   S_707.SPARE89 := FALSE;
   S_707.SPARE90 := FALSE;
   S_707.SPARE91 := FALSE;
   S_707.SPARE92 := FALSE;
   S_707.SPARE93 := FALSE;
   S_707.SPARE94 := FALSE;
   S_707.SPARE95 := FALSE;
   S_707.TL_DC_M_ADV_PB := FALSE;
   S_707.TL_DC_M_RET_PB := FALSE;
   S_707.SPARE98 := FALSE;
   S_707.SPARE99 := FALSE;
   S_707.SPARE100 := FALSE;
   S_707.SPARE101 := FALSE;
   S_707.SPARE102 := FALSE;
   S_707.SPARE103 := FALSE;
   S_707.SPARE104 := FALSE;
   S_707.SPARE105 := FALSE;
   S_707.SPARE106 := FALSE;
   S_707.SPARE107 := FALSE;
   S_707.SPARE108 := FALSE;
   S_707.SPARE109 := FALSE;
   S_707.SPARE110 := FALSE;
   S_707.SPARE111 := FALSE;
   S_707.SPARE112 := FALSE;
   S_707.SPARE113 := FALSE;
   S_707.SPARE114 := FALSE;
   S_707.SPARE115 := FALSE;
   S_707.SPARE116 := FALSE;
   S_707.SPARE117 := FALSE;
   S_707.SPARE118 := FALSE;
   S_707.SPARE119 := FALSE;
   S_707.SPARE120 := FALSE;
   S_707.SPARE121 := FALSE;
   S_707.SPARE122 := FALSE;
   S_707.SPARE123 := FALSE;
   S_707.SPARE124 := FALSE;
   S_707.SPARE125 := FALSE;
   S_707.SPARE126 := FALSE;
   S_707.SPARE127 := FALSE;
   S_707.SPARE128 := FALSE;
   S_707.SPARE129 := FALSE;
   S_707.SPARE130 := FALSE;
   S_707.SPARE131 := FALSE;
   S_707.SPARE132 := FALSE;
   S_707.SPARE133 := FALSE;
   S_707.SPARE134 := FALSE;
   S_707.SPARE135 := FALSE;
   S_707.SPARE136 := FALSE;
   S_707.SPARE137 := FALSE;
   S_707.SPARE138 := FALSE;
   S_707.SPARE139 := FALSE;
   S_707.SPARE140 := FALSE;
   S_707.SPARE141 := FALSE;
   S_707.SPARE142 := FALSE;
   S_707.SPARE143 := FALSE;
   S_707.SPARE144 := FALSE;
   S_707.SPARE145 := FALSE;
   S_707.SPARE146 := FALSE;
   S_707.SPARE147 := FALSE;
   S_707.SPARE148 := FALSE;
   S_707.SPARE149 := FALSE;
   S_707.SPARE150 := FALSE;
   S_707.SPARE151 := FALSE;
   S_707.SPARE152 := FALSE;
   S_707.SPARE153 := FALSE;
   S_707.SPARE154 := FALSE;
   S_707.SPARE155 := FALSE;
   S_707.SPARE156 := FALSE;
   S_707.SPARE157 := FALSE;
   S_707.SPARE158 := FALSE;
   S_707.SPARE159 := FALSE;
   S_707.SPARE160 := FALSE;
   S_707.SPARE161 := FALSE;
   S_707.HOOK_PIN_UP_LP := W#16#0;
   S_707.HOOK_PIN_DOWN_LP := W#16#700;
   S_707.DAECHA_LOCK_ADV_LP := W#16#300;
   S_707.DAECHA_LOCK_RET_LP := W#16#0;
   S_707.ELE_ADV_LP := W#16#300;
   S_707.ELE_RET_LP := W#16#0;
   S_707.AIR_ELE_ADV_LP := W#16#300;
   S_707.AIR_ELE_RET_LP := W#16#0;
   S_707.SP_WORD19 := W#16#0;
   S_707.SP_WORD20 := W#16#0;
   S_707.LM_DC_PIN_UP_LP := W#16#0;
   S_707.LM_DC_PIN_DOWN_LP := W#16#0;
   S_707.LM_DC_1ST_CLAMP1_ADV_LP := W#16#0;
   S_707.LM_DC_1ST_CLAMP1_RET_LP := W#16#0;
   S_707.LM_DC_1ST_CLAMP2_ADV_LP := W#16#0;
   S_707.LM_DC_1ST_CLAMP2_RET_LP := W#16#0;
   S_707.LM_DC_1ST_CLAMP3_ADV_LP := W#16#0;
   S_707.LM_DC_1ST_CLAMP3_RET_LP := W#16#0;
   S_707.LM_DC_1ST_CLAMP4_ADV_LP := W#16#0;
   S_707.LM_DC_1ST_CLAMP4_RET_LP := W#16#0;
   S_707.LM_DC_2ND_CLAMP1_ADV_LP := W#16#0;
   S_707.LM_DC_2ND_CLAMP1_RET_LP := W#16#0;
   S_707.LM_DC_2ND_CLAMP2_ADV_LP := W#16#0;
   S_707.LM_DC_2ND_CLAMP2_RET_LP := W#16#0;
   S_707.LM_DC_2ND_CLAMP3_ADV_LP := W#16#0;
   S_707.LM_DC_2ND_CLAMP3_RET_LP := W#16#0;
   S_707.LM_DC_2ND_CLAMP4_ADV_LP := W#16#0;
   S_707.LM_DC_2ND_CLAMP4_RET_LP := W#16#0;
   S_707.LM_DC_2ND_CLAMP5_ADV_LP := W#16#0;
   S_707.LM_DC_2ND_CLAMP5_RET_LP := W#16#0;
   S_707.LM_DC_DR_STK_PIN_UP_LP := W#16#0;
   S_707.LM_DC_DR_STK_PIN_DOWN_LP := W#16#0;
   S_707.LM_DC_OTR_CLAMP_ADV_LP := W#16#0;
   S_707.LM_DC_OTR_CLAMP_RET_LP := W#16#0;
   S_707.LM_DC_ASSY_CLAMP_ADV_LP := W#16#0;
   S_707.LM_DC_ASSY_CLAMP_RET_LP := W#16#0;
   S_707.LM_DC_FF_PIN_UP_LP := W#16#0;
   S_707.LM_DC_FF_PIN_DOWN_LP := W#16#0;
   S_707.LM_DC_FF_CLAMP_ADV_LP := W#16#0;
   S_707.LM_DC_FF_CLAMP_RET_LP := W#16#0;
   S_707.LM_DC_2ND_CLAMP6_ADV_LP := W#16#0;
   S_707.LM_DC_2ND_CLAMP6_RET_LP := W#16#0;
   S_707.LM_DC_2ND_CLAMP7_ADV_LP := W#16#0;
   S_707.LM_DC_2ND_CLAMP7_RET_LP := W#16#0;
   S_707.LM_DC_1ST_CLAMP5_ADV_LP := W#16#0;
   S_707.LM_DC_1ST_CLAMP5_RET_LP := W#16#0;
   S_707.SP_WORD68 := W#16#0;
   S_707.SP_WORD69 := W#16#0;
   S_707.SP_WORD70 := W#16#0;
   S_707.SP_WORD71 := W#16#0;
   S_707.TL_DC_PIN_UP_LP := W#16#F00;
   S_707.TL_DC_PIN_DOWN_LP := W#16#0;
   S_707.TL_DC_LATCH1_ADV_LP := W#16#3F00;
   S_707.TL_DC_LATCH1_RET_LP := W#16#0;
   S_707.TL_DC_LATCH2_ADV_LP := W#16#700;
   S_707.TL_DC_LATCH2_RET_LP := W#16#0;
   S_707.TL_DC_1ST_CLAMP1_ADV_LP := W#16#300;
   S_707.TL_DC_1ST_CLAMP1_RET_LP := W#16#0;
   S_707.TL_DC_1ST_CLAMP2_ADV_LP := W#16#300;
   S_707.TL_DC_1ST_CLAMP2_RET_LP := W#16#0;
   S_707.TL_DC_1ST_CLAMP3_ADV_LP := W#16#300;
   S_707.TL_DC_1ST_CLAMP3_RET_LP := W#16#0;
   S_707.TL_DC_2ND_CLAMP1_ADV_LP := W#16#300;
   S_707.TL_DC_2ND_CLAMP1_RET_LP := W#16#0;
   S_707.TL_DC_2ND_CLAMP2_ADV_LP := W#16#300;
   S_707.TL_DC_2ND_CLAMP2_RET_LP := W#16#0;
   S_707.TL_DC_U261_ADV_LP := W#16#300;
   S_707.TL_DC_U261_RET_LP := W#16#0;
   S_707.TL_DC_U261_CLAMP_ADV_LP := W#16#300;
   S_707.TL_DC_U261_CLAMP_RET_LP := W#16#0;
   S_707.TL_DC_U269_UP_LP := W#16#100;
   S_707.TL_DC_U269_DOWN_LP := W#16#0;
   S_707.TL_DC_U269_CLAMP_ADV_LP := W#16#300;
   S_707.TL_DC_U269_CLAMP_RET_LP := W#16#0;
   S_707.TL_DC_3RD_CLAMP_ADV_LP := W#16#100;
   S_707.TL_DC_3RD_CLAMP_RET_LP := W#16#0;
   S_707.TL_DC_U262_1_UP_LP := W#16#0;
   S_707.TL_DC_U262_1_DOWN_LP := W#16#300;
   S_707.TL_DC_U262_1_ADV_LP := W#16#0;
   S_707.TL_DC_U262_1_RET_LP := W#16#300;
   S_707.TL_DC_U262_1_CLP_ADV_LP := W#16#0;
   S_707.TL_DC_U262_1_CLP_RET_LP := W#16#300;
   S_707.TL_DC_U261_2_CLP_ADV_LP := W#16#0;
   S_707.TL_DC_U261_2_CLP_RET_LP := W#16#300;
   S_707.SP_WORD106 := W#16#0;
   S_707.SP_WORD107 := W#16#0;
   S_707.SP_WORD108 := W#16#0;
   S_707.SP_WORD109 := W#16#0;
   S_707.SP_WORD110 := W#16#0;
   S_707.SP_WORD111 := W#16#0;
   S_708.M_AUTO_SEL := FALSE;
   S_708.M_MANUAL_SEL := FALSE;
   S_708.M_READY_PB := FALSE;
   S_708.M_AUTO_RUN_PB := FALSE;
   S_708.M_WORK_COMP_SET_PB := FALSE;
   S_708.M_WORK_COMP_RST_PB := FALSE;
   S_708.M_HOME_POS_PB := FALSE;
   S_708.M_708_L_R_BT_ERR_RST := FALSE;
   S_708.HOOK_PIN_SEL := FALSE;
   S_708.EJECT_SEL := FALSE;
   S_708.SAFETY_PIN_SEL := FALSE;
   S_708.DAECHA_OUT_SEL := FALSE;
   S_708.ELE_UP_DN_SEL := FALSE;
   S_708.ELE_ADV_RET_SEL := FALSE;
   S_708.SPARE15 := FALSE;
   S_708.SPARE16 := FALSE;
   S_708.SPARE17 := FALSE;
   S_708.SPARE18 := FALSE;
   S_708.SPARE19 := FALSE;
   S_708.SPARE20 := FALSE;
   S_708.SPARE21 := FALSE;
   S_708.SPARE22 := FALSE;
   S_708.SPARE23 := FALSE;
   S_708.SPARE24 := FALSE;
   S_708.SPARE25 := FALSE;
   S_708.SPARE26 := FALSE;
   S_708.SPARE27 := FALSE;
   S_708.SPARE28 := FALSE;
   S_708.SPARE29 := FALSE;
   S_708.SPARE30 := FALSE;
   S_708.M_ADV_PB := FALSE;
   S_708.M_RET_PB := FALSE;
   S_708.LM_DC_PIN_SEL := FALSE;
   S_708.LM_DC_1ST_CLAMP1_SEL := FALSE;
   S_708.LM_DC_1ST_CLAMP2_SEL := FALSE;
   S_708.LM_DC_1ST_CLAMP3_SEL := FALSE;
   S_708.LM_DC_1ST_CLAMP4_SEL := FALSE;
   S_708.LM_DC_2ND_CLAMP1_SEL := FALSE;
   S_708.LM_DC_2ND_CLAMP2_SEL := FALSE;
   S_708.LM_DC_2ND_CLAMP3_SEL := FALSE;
   S_708.LM_DC_2ND_CLAMP4_SEL := FALSE;
   S_708.LM_DC_2ND_CLAMP5_SEL := FALSE;
   S_708.LM_DC_DR_STK_PIN_SEL := FALSE;
   S_708.LM_DC_OTR_CLAMP_SEL := FALSE;
   S_708.LM_DC_ASSY_CLAMP_SEL := FALSE;
   S_708.LM_DC_FF_PIN_SEL := FALSE;
   S_708.LM_DC_FF_CLAMP_SEL := FALSE;
   S_708.LM_DC_2ND_CLAMP6_SEL := FALSE;
   S_708.SPARE50 := FALSE;
   S_708.SPARE51 := FALSE;
   S_708.SPARE52 := FALSE;
   S_708.SPARE53 := FALSE;
   S_708.SPARE54 := FALSE;
   S_708.SPARE55 := FALSE;
   S_708.SPARE56 := FALSE;
   S_708.SPARE57 := FALSE;
   S_708.SPARE58 := FALSE;
   S_708.SPARE59 := FALSE;
   S_708.SPARE60 := FALSE;
   S_708.SPARE61 := FALSE;
   S_708.SPARE62 := FALSE;
   S_708.SPARE63 := FALSE;
   S_708.LM_DC_M_ADV_PB := FALSE;
   S_708.LM_DC_M_RET_PB := FALSE;
   S_708.TL_DC_PIN_SEL := FALSE;
   S_708.TL_DC_LATCH1_SEL := FALSE;
   S_708.TL_DC_1ST_CLAMP_SEL := FALSE;
   S_708.TL_DC_2ND_CLAMP_SEL := FALSE;
   S_708.TL_DC_U261_SEL := FALSE;
   S_708.TL_DC_U261_CLAMP_SEL := FALSE;
   S_708.TL_DC_U269_UP_DN_SEL := FALSE;
   S_708.TL_DC_U269_CLAMP_SEL := FALSE;
   S_708.TL_DC_3RD_CLAMP_SEL := FALSE;
   S_708.TL_DC_U262_1_UP_DN_SEL := FALSE;
   S_708.TL_DC_U262_1_SEL := FALSE;
   S_708.TL_DC_U262_1_CLAMP_SEL := FALSE;
   S_708.TL_DC_U261_2_CLAMP_SEL := FALSE;
   S_708.SPARE79 := FALSE;
   S_708.SPARE80 := FALSE;
   S_708.SPARE81 := FALSE;
   S_708.SPARE82 := FALSE;
   S_708.SPARE83 := FALSE;
   S_708.SPARE84 := FALSE;
   S_708.SPARE85 := FALSE;
   S_708.SPARE86 := FALSE;
   S_708.SPARE87 := FALSE;
   S_708.SPARE88 := FALSE;
   S_708.SPARE89 := FALSE;
   S_708.SPARE90 := FALSE;
   S_708.SPARE91 := FALSE;
   S_708.SPARE92 := FALSE;
   S_708.SPARE93 := FALSE;
   S_708.SPARE94 := FALSE;
   S_708.SPARE95 := FALSE;
   S_708.TL_DC_M_ADV_PB := FALSE;
   S_708.TL_DC_M_RET_PB := FALSE;
   S_708.SPARE98 := FALSE;
   S_708.SPARE99 := FALSE;
   S_708.SPARE100 := FALSE;
   S_708.SPARE101 := FALSE;
   S_708.SPARE102 := FALSE;
   S_708.SPARE103 := FALSE;
   S_708.SPARE104 := FALSE;
   S_708.SPARE105 := FALSE;
   S_708.SPARE106 := FALSE;
   S_708.SPARE107 := FALSE;
   S_708.SPARE108 := FALSE;
   S_708.SPARE109 := FALSE;
   S_708.SPARE110 := FALSE;
   S_708.SPARE111 := FALSE;
   S_708.SPARE112 := FALSE;
   S_708.SPARE113 := FALSE;
   S_708.SPARE114 := FALSE;
   S_708.SPARE115 := FALSE;
   S_708.SPARE116 := FALSE;
   S_708.SPARE117 := FALSE;
   S_708.SPARE118 := FALSE;
   S_708.SPARE119 := FALSE;
   S_708.SPARE120 := FALSE;
   S_708.SPARE121 := FALSE;
   S_708.SPARE122 := FALSE;
   S_708.SPARE123 := FALSE;
   S_708.SPARE124 := FALSE;
   S_708.SPARE125 := FALSE;
   S_708.SPARE126 := FALSE;
   S_708.SPARE127 := FALSE;
   S_708.SPARE128 := FALSE;
   S_708.SPARE129 := FALSE;
   S_708.ELE_AR_ADV_LP := W#16#300;
   S_708.ELE_AR_RET_LP := W#16#0;
   S_708.HOOK_PIN_UP_LP := W#16#0;
   S_708.HOOK_PIN_DOWN_LP := W#16#300;
   S_708.EJECT_UP_LP := W#16#0;
   S_708.EJECT_DOWN_LP := W#16#300;
   S_708.SAFETY_PIN_UP_LP := W#16#300;
   S_708.SAFETY_PIN_UDOWN_LP := W#16#0;
   S_708.DAECHA_OUT_ADV_LP := W#16#0;
   S_708.DAECHA_OUT_RET_LP := W#16#0;
   S_708.ELE_UD_UP_LP := W#16#300;
   S_708.ELE_UD_DOWN_LP := W#16#0;
   S_708.LM_DC_PIN_UP_LP := W#16#0;
   S_708.LM_DC_PIN_DOWN_LP := W#16#0;
   S_708.LM_DC_1ST_CLAMP1_ADV_LP := W#16#0;
   S_708.LM_DC_1ST_CLAMP1_RET_LP := W#16#0;
   S_708.LM_DC_1ST_CLAMP2_ADV_LP := W#16#0;
   S_708.LM_DC_1ST_CLAMP2_RET_LP := W#16#0;
   S_708.LM_DC_1ST_CLAMP3_ADV_LP := W#16#0;
   S_708.LM_DC_1ST_CLAMP3_RET_LP := W#16#0;
   S_708.LM_DC_1ST_CLAMP4_ADV_LP := W#16#0;
   S_708.LM_DC_1ST_CLAMP4_RET_LP := W#16#0;
   S_708.LM_DC_2ND_CLAMP1_ADV_LP := W#16#0;
   S_708.LM_DC_2ND_CLAMP1_RET_LP := W#16#0;
   S_708.LM_DC_2ND_CLAMP2_ADV_LP := W#16#0;
   S_708.LM_DC_2ND_CLAMP2_RET_LP := W#16#0;
   S_708.LM_DC_2ND_CLAMP3_ADV_LP := W#16#0;
   S_708.LM_DC_2ND_CLAMP3_RET_LP := W#16#0;
   S_708.LM_DC_2ND_CLAMP4_ADV_LP := W#16#0;
   S_708.LM_DC_2ND_CLAMP4_RET_LP := W#16#0;
   S_708.LM_DC_2ND_CLAMP5_ADV_LP := W#16#0;
   S_708.LM_DC_2ND_CLAMP5_RET_LP := W#16#0;
   S_708.LM_DC_DR_STK_PIN_UP_LP := W#16#0;
   S_708.LM_DC_DR_STK_PIN_DOWN_LP := W#16#0;
   S_708.LM_DC_OTR_CLAMP_ADV_LP := W#16#0;
   S_708.LM_DC_OTR_CLAMP_RET_LP := W#16#0;
   S_708.LM_DC_ASSY_CLAMP_ADV_LP := W#16#0;
   S_708.LM_DC_ASSY_CLAMP_RET_LP := W#16#0;
   S_708.LM_DC_FF_PIN_UP_LP := W#16#0;
   S_708.LM_DC_FF_PIN_DOWN_LP := W#16#0;
   S_708.LM_DC_FF_CLAMP_ADV_LP := W#16#0;
   S_708.LM_DC_FF_CLAMP_RET_LP := W#16#0;
   S_708.LM_DC_2ND_CLAMP6_ADV_LP := W#16#0;
   S_708.LM_DC_2ND_CLAMP6_RET_LP := W#16#0;
   S_708.LM_DC_2ND_CLAMP7_ADV_LP := W#16#0;
   S_708.LM_DC_2ND_CLAMP7_RET_LP := W#16#0;
   S_708.LM_DC_1ST_CLAMP5_ADV_LP := W#16#0;
   S_708.LM_DC_1ST_CLAMP5_RET_LP := W#16#0;
   S_708.SP_WORD68 := W#16#0;
   S_708.SP_WORD69 := W#16#0;
   S_708.SP_WORD70 := W#16#0;
   S_708.SP_WORD71 := W#16#0;
   S_708.TL_DC_PIN_UP_LP := W#16#0;
   S_708.TL_DC_PIN_DOWN_LP := W#16#F00;
   S_708.TL_DC_LATCH1_ADV_LP := W#16#0;
   S_708.TL_DC_LATCH1_RET_LP := W#16#3F00;
   S_708.TL_DC_LATCH2_ADV_LP := W#16#0;
   S_708.TL_DC_LATCH2_RET_LP := W#16#700;
   S_708.TL_DC_1ST_CLAMP1_ADV_LP := W#16#0;
   S_708.TL_DC_1ST_CLAMP1_RET_LP := W#16#3F00;
   S_708.TL_DC_1ST_CLAMP2_ADV_LP := W#16#0;
   S_708.TL_DC_1ST_CLAMP2_RET_LP := W#16#3F00;
   S_708.TL_DC_1ST_CLAMP3_ADV_LP := W#16#0;
   S_708.TL_DC_1ST_CLAMP3_RET_LP := W#16#F00;
   S_708.TL_DC_2ND_CLAMP1_ADV_LP := W#16#0;
   S_708.TL_DC_2ND_CLAMP1_RET_LP := W#16#3F00;
   S_708.TL_DC_2ND_CLAMP2_ADV_LP := W#16#0;
   S_708.TL_DC_2ND_CLAMP2_RET_LP := W#16#3F00;
   S_708.TL_DC_U261_ADV_LP := W#16#0;
   S_708.TL_DC_U261_RET_LP := W#16#300;
   S_708.TL_DC_U261_CLAMP_ADV_LP := W#16#0;
   S_708.TL_DC_U261_CLAMP_RET_LP := W#16#300;
   S_708.TL_DC_U269_UP_LP := W#16#0;
   S_708.TL_DC_U269_DOWN_LP := W#16#300;
   S_708.TL_DC_U269_CLAMP_ADV_LP := W#16#0;
   S_708.TL_DC_U269_CLAMP_RET_LP := W#16#700;
   S_708.TL_DC_3RD_CLAMP_ADV_LP := W#16#0;
   S_708.TL_DC_3RD_CLAMP_RET_LP := W#16#300;
   S_708.TL_DC_U262_1_UP_LP := W#16#0;
   S_708.TL_DC_U262_1_DOWN_LP := W#16#300;
   S_708.TL_DC_U262_1_ADV_LP := W#16#0;
   S_708.TL_DC_U262_1_RET_LP := W#16#300;
   S_708.TL_DC_U262_1_CLP_ADV_LP := W#16#0;
   S_708.TL_DC_U262_1_CLP_RET_LP := W#16#300;
   S_708.TL_DC_U261_2_CLP_ADV_LP := W#16#0;
   S_708.TL_DC_U261_2_CLP_RET_LP := W#16#300;
   S_708.SP_WORD106 := W#16#0;
   S_708.SP_WORD107 := W#16#0;
   S_708.SP_WORD108 := W#16#0;
   S_708.SP_WORD109 := W#16#0;
   S_708.AIR_ELE_AR_ADV_LP := W#16#300;
   S_708.AIR_ELE_AR_RET_LP := W#16#0;
   S_UPDL.M_AUTO_SEL := FALSE;
   S_UPDL.M_MANUAL_SEL := FALSE;
   S_UPDL.M_READY_PB := FALSE;
   S_UPDL.M_AUTO_RUN_PB := FALSE;
   S_UPDL.M_WORK_COMP_SET_PB := FALSE;
   S_UPDL.M_WORK_COMP_RST_PB := FALSE;
   S_UPDL.M_HOME_POS_PB := FALSE;
   S_UPDL.SPARE8 := FALSE;
   S_UPDL.DAECHA_CLAMP_SEL := FALSE;
   S_UPDL.ELE_AIR_UP_DN_SEL := FALSE;
   S_UPDL.ELE_AIR_ADV_RET_SEL := FALSE;
   S_UPDL.DAECHA_IN_SEL := TRUE;
   S_UPDL.DAECHA_OUT_SEL := FALSE;
   S_UPDL.LIFT_LOCK_SEL := FALSE;
   S_UPDL.LIFT_UP_DN_SEL := FALSE;
   S_UPDL.SPARE16 := FALSE;
   S_UPDL.SPARE17 := FALSE;
   S_UPDL.SPARE18 := FALSE;
   S_UPDL.SPARE19 := FALSE;
   S_UPDL.SPARE20 := FALSE;
   S_UPDL.SPARE21 := FALSE;
   S_UPDL.SPARE22 := FALSE;
   S_UPDL.SPARE23 := FALSE;
   S_UPDL.SPARE24 := FALSE;
   S_UPDL.SPARE25 := FALSE;
   S_UPDL.SPARE26 := FALSE;
   S_UPDL.SPARE27 := FALSE;
   S_UPDL.SPARE28 := FALSE;
   S_UPDL.SPARE29 := FALSE;
   S_UPDL.SPARE30 := FALSE;
   S_UPDL.M_ADV_PB := FALSE;
   S_UPDL.M_RET_PB := FALSE;
   S_UPDL.SPARE34 := FALSE;
   S_UPDL.SPARE35 := FALSE;
   S_UPDL.SPARE36 := FALSE;
   S_UPDL.SPARE37 := FALSE;
   S_UPDL.SPARE38 := FALSE;
   S_UPDL.SPARE39 := FALSE;
   S_UPDL.SPARE40 := FALSE;
   S_UPDL.SPARE41 := FALSE;
   S_UPDL.SPARE42 := FALSE;
   S_UPDL.SPARE43 := FALSE;
   S_UPDL.SPARE44 := FALSE;
   S_UPDL.SPARE45 := FALSE;
   S_UPDL.SPARE46 := FALSE;
   S_UPDL.SPARE47 := FALSE;
   S_UPDL.SPARE48 := FALSE;
   S_UPDL.SPARE49 := FALSE;
   S_UPDL.SPARE50 := FALSE;
   S_UPDL.SPARE51 := FALSE;
   S_UPDL.SPARE52 := FALSE;
   S_UPDL.SPARE53 := FALSE;
   S_UPDL.SPARE54 := FALSE;
   S_UPDL.SPARE55 := FALSE;
   S_UPDL.SPARE56 := FALSE;
   S_UPDL.SPARE57 := FALSE;
   S_UPDL.SPARE58 := FALSE;
   S_UPDL.SPARE59 := FALSE;
   S_UPDL.SPARE60 := FALSE;
   S_UPDL.SPARE61 := FALSE;
   S_UPDL.SPARE62 := FALSE;
   S_UPDL.SPARE63 := FALSE;
   S_UPDL.SPARE64 := FALSE;
   S_UPDL.SPARE65 := FALSE;
   S_UPDL.SPARE66 := FALSE;
   S_UPDL.SPARE67 := FALSE;
   S_UPDL.SPARE68 := FALSE;
   S_UPDL.SPARE69 := FALSE;
   S_UPDL.SPARE70 := FALSE;
   S_UPDL.SPARE71 := FALSE;
   S_UPDL.SPARE72 := FALSE;
   S_UPDL.SPARE73 := FALSE;
   S_UPDL.SPARE74 := FALSE;
   S_UPDL.SPARE75 := FALSE;
   S_UPDL.SPARE76 := FALSE;
   S_UPDL.SPARE77 := FALSE;
   S_UPDL.SPARE78 := FALSE;
   S_UPDL.SPARE79 := FALSE;
   S_UPDL.SPARE80 := FALSE;
   S_UPDL.SPARE81 := FALSE;
   S_UPDL.SPARE82 := FALSE;
   S_UPDL.SPARE83 := FALSE;
   S_UPDL.SPARE84 := FALSE;
   S_UPDL.SPARE85 := FALSE;
   S_UPDL.SPARE86 := FALSE;
   S_UPDL.SPARE87 := FALSE;
   S_UPDL.SPARE88 := FALSE;
   S_UPDL.SPARE89 := FALSE;
   S_UPDL.SPARE90 := FALSE;
   S_UPDL.SPARE91 := FALSE;
   S_UPDL.SPARE92 := FALSE;
   S_UPDL.SPARE93 := FALSE;
   S_UPDL.SPARE94 := FALSE;
   S_UPDL.SPARE95 := FALSE;
   S_UPDL.SPARE96 := FALSE;
   S_UPDL.SPARE97 := FALSE;
   S_UPDL.SPARE98 := FALSE;
   S_UPDL.SPARE99 := FALSE;
   S_UPDL.SPARE100 := FALSE;
   S_UPDL.SPARE101 := FALSE;
   S_UPDL.SPARE102 := FALSE;
   S_UPDL.SPARE103 := FALSE;
   S_UPDL.SPARE104 := FALSE;
   S_UPDL.SPARE105 := FALSE;
   S_UPDL.SPARE106 := FALSE;
   S_UPDL.SPARE107 := FALSE;
   S_UPDL.SPARE108 := FALSE;
   S_UPDL.SPARE109 := FALSE;
   S_UPDL.SPARE110 := FALSE;
   S_UPDL.SPARE111 := FALSE;
   S_UPDL.SPARE112 := FALSE;
   S_UPDL.SPARE113 := FALSE;
   S_UPDL.SPARE114 := FALSE;
   S_UPDL.SPARE115 := FALSE;
   S_UPDL.SPARE116 := FALSE;
   S_UPDL.SPARE117 := FALSE;
   S_UPDL.SPARE118 := FALSE;
   S_UPDL.SPARE119 := FALSE;
   S_UPDL.SPARE120 := FALSE;
   S_UPDL.SPARE121 := FALSE;
   S_UPDL.SPARE122 := FALSE;
   S_UPDL.SPARE123 := FALSE;
   S_UPDL.SPARE124 := FALSE;
   S_UPDL.SPARE125 := FALSE;
   S_UPDL.SPARE126 := FALSE;
   S_UPDL.SPARE127 := FALSE;
   S_UPDL.SPARE128 := FALSE;
   S_UPDL.SPARE129 := FALSE;
   S_UPDL.SPARE130 := FALSE;
   S_UPDL.SPARE131 := FALSE;
   S_UPDL.SPARE132 := FALSE;
   S_UPDL.SPARE133 := FALSE;
   S_UPDL.SPARE134 := FALSE;
   S_UPDL.SPARE135 := FALSE;
   S_UPDL.SPARE136 := FALSE;
   S_UPDL.SPARE137 := FALSE;
   S_UPDL.SPARE138 := FALSE;
   S_UPDL.SPARE139 := FALSE;
   S_UPDL.SPARE140 := FALSE;
   S_UPDL.SPARE141 := FALSE;
   S_UPDL.SPARE142 := FALSE;
   S_UPDL.SPARE143 := FALSE;
   S_UPDL.SPARE144 := FALSE;
   S_UPDL.SPARE145 := FALSE;
   S_UPDL.SPARE146 := FALSE;
   S_UPDL.SPARE147 := FALSE;
   S_UPDL.SPARE148 := FALSE;
   S_UPDL.SPARE149 := FALSE;
   S_UPDL.SPARE150 := FALSE;
   S_UPDL.SPARE151 := FALSE;
   S_UPDL.SPARE152 := FALSE;
   S_UPDL.SPARE153 := FALSE;
   S_UPDL.SPARE154 := FALSE;
   S_UPDL.SPARE155 := FALSE;
   S_UPDL.SPARE156 := FALSE;
   S_UPDL.SPARE157 := FALSE;
   S_UPDL.SPARE158 := FALSE;
   S_UPDL.SPARE159 := FALSE;
   S_UPDL.SPARE160 := FALSE;
   S_UPDL.SPARE161 := FALSE;
   S_UPDL.DAECHA_CLAMP_ADV_LP := W#16#0;
   S_UPDL.DAECHA_CLAMP_RET_LP := W#16#700;
   S_UPDL.ELE_AIR_UP_DN_UP_LP := W#16#0;
   S_UPDL.ELE_AIR_UP_DN_DOWN_LP := W#16#300;
   S_UPDL.ELE_AIR_ADV_RET_ADV_LP := W#16#0;
   S_UPDL.ELE_AIR_ADV_RET_RET_LP := W#16#300;
   S_UPDL.DAECHA_IN_ADV_LP := W#16#0;
   S_UPDL.DAECHA_IN_RET_LP := W#16#0;
   S_UPDL.DAECHA_OUT_ADV_LP := W#16#0;
   S_UPDL.DAECHA_OUT_RET_LP := W#16#0;
   S_UPDL.LIFT_LOCL_ADV_LP := W#16#700;
   S_UPDL.LIFT_LOCL_RET_LP := W#16#0;
   S_UPDL.LIFT_UP_DN_UP_LP := W#16#300;
   S_UPDL.LIFT_UP_DN_DOWN_LP := W#16#0;
   S_UPDL.SP_WORD25 := W#16#0;
   S_UPDL.SP_WORD26 := W#16#0;
   S_UPDL.SP_WORD27 := W#16#0;
   S_UPDL.SP_WORD28 := W#16#0;
   S_UPDL.SP_WORD29 := W#16#0;
   S_UPDL.SP_WORD30 := W#16#0;
   S_UPDL.SP_WORD31 := W#16#0;
   S_UPDL.SP_WORD32 := W#16#0;
   S_UPDL.SP_WORD33 := W#16#0;
   S_UPDL.SP_WORD34 := W#16#0;
   S_UPDL.SP_WORD35 := W#16#0;
   S_UPDL.SP_WORD36 := W#16#0;
   S_UPDL.SP_WORD37 := W#16#0;
   S_UPDL.SP_WORD38 := W#16#0;
   S_UPDL.SP_WORD39 := W#16#0;
   S_UPDL.SP_WORD40 := W#16#0;
   S_UPDL.SP_WORD41 := W#16#0;
   S_UPDL.SP_WORD42 := W#16#0;
   S_UPDL.SP_WORD43 := W#16#0;
   S_UPDL.SP_WORD44 := W#16#0;
   S_UPDL.SP_WORD45 := W#16#0;
   S_UPDL.SP_WORD46 := W#16#0;
   S_UPDL.SP_WORD47 := W#16#0;
   S_UPDL.SP_WORD49 := W#16#0;
   S_UPDL.SP_WORD50 := W#16#0;
   S_UPDL.SP_WORD51 := W#16#0;
   S_UPDL.SP_WORD52 := W#16#0;
   S_UPDL.SP_WORD53 := W#16#0;
   S_UPDL.SP_WORD54 := W#16#0;
   S_UPDL.SP_WORD55 := W#16#0;
   S_UPDL.SP_WORD56 := W#16#0;
   S_UPDL.SP_WORD57 := W#16#0;
   S_UPDL.SP_WORD58 := W#16#0;
   S_UPDL.SP_WORD59 := W#16#0;
   S_UPDL.SP_WORD60 := W#16#0;
   S_UPDL.SP_WORD61 := W#16#0;
   S_UPDL.SP_WORD62 := W#16#0;
   S_UPDL.SP_WORD63 := W#16#0;
   S_UPDL.SP_WORD64 := W#16#0;
   S_UPDL.SP_WORD65 := W#16#0;
   S_UPDL.SP_WORD66 := W#16#0;
   S_UPDL.SP_WORD67 := W#16#0;
   S_UPDL.SP_WORD68 := W#16#0;
   S_UPDL.SP_WORD69 := W#16#0;
   S_UPDL.SP_WORD70 := W#16#0;
   S_UPDL.SP_WORD71 := W#16#0;
   S_UPDL.SP_WORD72 := W#16#0;
   S_UPDL.SP_WORD73 := W#16#0;
   S_UPDL.SP_WORD74 := W#16#0;
   S_UPDL.SP_WORD75 := W#16#0;
   S_UPDL.SP_WORD76 := W#16#0;
   S_UPDL.SP_WORD77 := W#16#0;
   S_UPDL.SP_WORD78 := W#16#0;
   S_UPDL.SP_WORD79 := W#16#0;
   S_UPDL.SP_WORD80 := W#16#0;
   S_UPDL.SP_WORD81 := W#16#0;
   S_UPDL.SP_WORD82 := W#16#0;
   S_UPDL.SP_WORD83 := W#16#0;
   S_UPDL.SP_WORD84 := W#16#0;
   S_UPDL.SP_WORD85 := W#16#0;
   S_UPDL.SP_WORD86 := W#16#0;
   S_UPDL.SP_WORD87 := W#16#0;
   S_UPDL.SP_WORD88 := W#16#0;
   S_UPDL.SP_WORD89 := W#16#0;
   S_UPDL.SP_WORD90 := W#16#0;
   S_UPDL.SP_WORD91 := W#16#0;
   S_UPDL.SP_WORD92 := W#16#0;
   S_UPDL.SP_WORD93 := W#16#0;
   S_UPDL.SP_WORD94 := W#16#0;
   S_UPDL.SP_WORD95 := W#16#0;
   S_UPDL.SP_WORD96 := W#16#0;
   S_UPDL.SP_WORD97 := W#16#0;
   S_UPDL.SP_WORD98 := W#16#0;
   S_UPDL.SP_WORD99 := W#16#0;
   S_UPDL.SP_WORD100 := W#16#0;
   S_UPDL.SP_WORD101 := W#16#0;
END_DATA_BLOCK

DATA_BLOCK DB 54
TITLE =
VERSION : 0.1


  STRUCT
   DP_1 : STRUCT 	//Temporary placeholder variable
    CHECK_ACTIVE : BOOL ;
    DATA_FIELD : ARRAY  [0 .. 54 ] OF BYTE ;
    SUM_SLAVE_DIAG : INT ;
    LIST_NOT_PRESENT : ARRAY  [0 .. 3 ] OF DWORD ;
    LIST_ERROR : ARRAY  [0 .. 3 ] OF DWORD ;
    RET_VALUE : INT ;
    DIAG_EVENT : BOOL ;
    STATION_ERR : BOOL ;
    RESTART : BOOL ;
    BUSY : BOOL ;
    SP1 : WORD ;
    SP2 : WORD ;
   END_STRUCT ;
   DP_2 : STRUCT 	//Temporary placeholder variable
    CHECK_ACTIVE : BOOL ;
    DATA_FIELD : ARRAY  [0 .. 54 ] OF BYTE ;
    SUM_SLAVE_DIAG : INT ;
    LIST_NOT_PRESENT : ARRAY  [0 .. 3 ] OF DWORD ;
    LIST_ERROR : ARRAY  [0 .. 3 ] OF DWORD ;
    RET_VALUE : INT ;
    DIAG_EVENT : BOOL ;
    STATION_ERR : BOOL ;
    RESTART : BOOL ;
    BUSY : BOOL ;
    SP1 : WORD ;
    SP2 : WORD ;
   END_STRUCT ;
   DP_3 : STRUCT 	//Temporary placeholder variable
    NDR : BOOL ;
    ERR : BOOL ;
    SP21 : ARRAY  [0 .. 3 ] OF WORD ;
    STATUS : WORD ;
    SP22 : WORD ;
    DIAGLNG : BYTE ;
    SP23 : ARRAY  [0 .. 3 ] OF BYTE ;
    LIST_ERROR : ARRAY  [0 .. 3 ] OF DWORD ;
    SP24 : ARRAY  [0 .. 12 ] OF BYTE ;
   END_STRUCT ;
   DP_4 : STRUCT 	//Temporary placeholder variable
    NDR : BOOL ;
    ERR : BOOL ;
    SP21 : ARRAY  [0 .. 3 ] OF WORD ;
    STATUS : WORD ;
    SP22 : WORD ;
    DIAGLNG : BYTE ;
    SP23 : ARRAY  [0 .. 3 ] OF BYTE ;
    LIST_ERROR : ARRAY  [0 .. 3 ] OF DWORD ;
    SP24 : ARRAY  [0 .. 12 ] OF BYTE ;
   END_STRUCT ;
   DP_5 : STRUCT 	//Temporary placeholder variable
    NDR : BOOL ;
    ERR : BOOL ;
    SP21 : ARRAY  [0 .. 3 ] OF WORD ;
    STATUS : WORD ;
    SP22 : WORD ;
    DIAGLNG : BYTE ;
    SP23 : ARRAY  [0 .. 3 ] OF BYTE ;
    LIST_ERROR : ARRAY  [0 .. 3 ] OF DWORD ;
    SP24 : ARRAY  [0 .. 12 ] OF BYTE ;
   END_STRUCT ;
   DP_6 : STRUCT 	//Temporary placeholder variable
    NDR : BOOL ;
    ERR : BOOL ;
    SP21 : ARRAY  [0 .. 3 ] OF WORD ;
    STATUS : WORD ;
    SP22 : WORD ;
    DIAGLNG : BYTE ;
    SP23 : ARRAY  [0 .. 3 ] OF BYTE ;
    LIST_ERROR : ARRAY  [0 .. 3 ] OF DWORD ;
    SP24 : ARRAY  [0 .. 12 ] OF BYTE ;
   END_STRUCT ;
   DP_7 : STRUCT 	//Temporary placeholder variable
    NDR : BOOL ;
    ERR : BOOL ;
    SP21 : ARRAY  [0 .. 3 ] OF WORD ;
    STATUS : WORD ;
    SP22 : WORD ;
    DIAGLNG : BYTE ;
    SP23 : ARRAY  [0 .. 3 ] OF BYTE ;
    LIST_ERROR : ARRAY  [0 .. 3 ] OF DWORD ;
    SP24 : ARRAY  [0 .. 12 ] OF BYTE ;
   END_STRUCT ;
   DP_8 : STRUCT 	//Temporary placeholder variable
    NDR : BOOL ;
    ERR : BOOL ;
    SP21 : ARRAY  [0 .. 3 ] OF WORD ;
    STATUS : WORD ;
    SP22 : WORD ;
    DIAGLNG : BYTE ;
    SP23 : ARRAY  [0 .. 3 ] OF BYTE ;
    LIST_ERROR : ARRAY  [0 .. 3 ] OF DWORD ;
    SP24 : ARRAY  [0 .. 12 ] OF BYTE ;
   END_STRUCT ;
   DP_9 : STRUCT 	//Temporary placeholder variable
    NDR : BOOL ;
    ERR : BOOL ;
    SP21 : ARRAY  [0 .. 3 ] OF WORD ;
    STATUS : WORD ;
    SP22 : WORD ;
    DIAGLNG : BYTE ;
    SP23 : ARRAY  [0 .. 3 ] OF BYTE ;
    LIST_ERROR : ARRAY  [0 .. 3 ] OF DWORD ;
    SP24 : ARRAY  [0 .. 12 ] OF BYTE ;
   END_STRUCT ;
   DP_10 : STRUCT 	//Temporary placeholder variable
    NDR : BOOL ;
    ERR : BOOL ;
    SP21 : ARRAY  [0 .. 3 ] OF WORD ;
    STATUS : WORD ;
    SP22 : WORD ;
    DIAGLNG : BYTE ;
    SP23 : ARRAY  [0 .. 3 ] OF BYTE ;
    LIST_ERROR : ARRAY  [0 .. 3 ] OF DWORD ;
    SP24 : ARRAY  [0 .. 12 ] OF BYTE ;
   END_STRUCT ;
  END_STRUCT ;
BEGIN
   DP_1.CHECK_ACTIVE := FALSE;
   DP_1.DATA_FIELD[0] := B#16#0;
   DP_1.DATA_FIELD[1] := B#16#0;
   DP_1.DATA_FIELD[2] := B#16#0;
   DP_1.DATA_FIELD[3] := B#16#0;
   DP_1.DATA_FIELD[4] := B#16#0;
   DP_1.DATA_FIELD[5] := B#16#0;
   DP_1.DATA_FIELD[6] := B#16#0;
   DP_1.DATA_FIELD[7] := B#16#0;
   DP_1.DATA_FIELD[8] := B#16#0;
   DP_1.DATA_FIELD[9] := B#16#0;
   DP_1.DATA_FIELD[10] := B#16#0;
   DP_1.DATA_FIELD[11] := B#16#0;
   DP_1.DATA_FIELD[12] := B#16#0;
   DP_1.DATA_FIELD[13] := B#16#0;
   DP_1.DATA_FIELD[14] := B#16#0;
   DP_1.DATA_FIELD[15] := B#16#0;
   DP_1.DATA_FIELD[16] := B#16#0;
   DP_1.DATA_FIELD[17] := B#16#0;
   DP_1.DATA_FIELD[18] := B#16#0;
   DP_1.DATA_FIELD[19] := B#16#0;
   DP_1.DATA_FIELD[20] := B#16#0;
   DP_1.DATA_FIELD[21] := B#16#0;
   DP_1.DATA_FIELD[22] := B#16#0;
   DP_1.DATA_FIELD[23] := B#16#0;
   DP_1.DATA_FIELD[24] := B#16#0;
   DP_1.DATA_FIELD[25] := B#16#0;
   DP_1.DATA_FIELD[26] := B#16#0;
   DP_1.DATA_FIELD[27] := B#16#0;
   DP_1.DATA_FIELD[28] := B#16#0;
   DP_1.DATA_FIELD[29] := B#16#0;
   DP_1.DATA_FIELD[30] := B#16#0;
   DP_1.DATA_FIELD[31] := B#16#0;
   DP_1.DATA_FIELD[32] := B#16#0;
   DP_1.DATA_FIELD[33] := B#16#0;
   DP_1.DATA_FIELD[34] := B#16#0;
   DP_1.DATA_FIELD[35] := B#16#0;
   DP_1.DATA_FIELD[36] := B#16#0;
   DP_1.DATA_FIELD[37] := B#16#0;
   DP_1.DATA_FIELD[38] := B#16#0;
   DP_1.DATA_FIELD[39] := B#16#0;
   DP_1.DATA_FIELD[40] := B#16#0;
   DP_1.DATA_FIELD[41] := B#16#0;
   DP_1.DATA_FIELD[42] := B#16#0;
   DP_1.DATA_FIELD[43] := B#16#0;
   DP_1.DATA_FIELD[44] := B#16#0;
   DP_1.DATA_FIELD[45] := B#16#0;
   DP_1.DATA_FIELD[46] := B#16#0;
   DP_1.DATA_FIELD[47] := B#16#0;
   DP_1.DATA_FIELD[48] := B#16#0;
   DP_1.DATA_FIELD[49] := B#16#0;
   DP_1.DATA_FIELD[50] := B#16#0;
   DP_1.DATA_FIELD[51] := B#16#0;
   DP_1.DATA_FIELD[52] := B#16#0;
   DP_1.DATA_FIELD[53] := B#16#0;
   DP_1.DATA_FIELD[54] := B#16#0;
   DP_1.SUM_SLAVE_DIAG := 0;
   DP_1.LIST_NOT_PRESENT[0] := DW#16#0;
   DP_1.LIST_NOT_PRESENT[1] := DW#16#0;
   DP_1.LIST_NOT_PRESENT[2] := DW#16#0;
   DP_1.LIST_NOT_PRESENT[3] := DW#16#0;
   DP_1.LIST_ERROR[0] := DW#16#0;
   DP_1.LIST_ERROR[1] := DW#16#0;
   DP_1.LIST_ERROR[2] := DW#16#0;
   DP_1.LIST_ERROR[3] := DW#16#0;
   DP_1.RET_VALUE := 0;
   DP_1.DIAG_EVENT := FALSE;
   DP_1.STATION_ERR := FALSE;
   DP_1.RESTART := FALSE;
   DP_1.BUSY := FALSE;
   DP_1.SP1 := W#16#0;
   DP_1.SP2 := W#16#0;
   DP_2.CHECK_ACTIVE := FALSE;
   DP_2.DATA_FIELD[0] := B#16#0;
   DP_2.DATA_FIELD[1] := B#16#0;
   DP_2.DATA_FIELD[2] := B#16#0;
   DP_2.DATA_FIELD[3] := B#16#0;
   DP_2.DATA_FIELD[4] := B#16#0;
   DP_2.DATA_FIELD[5] := B#16#0;
   DP_2.DATA_FIELD[6] := B#16#0;
   DP_2.DATA_FIELD[7] := B#16#0;
   DP_2.DATA_FIELD[8] := B#16#0;
   DP_2.DATA_FIELD[9] := B#16#0;
   DP_2.DATA_FIELD[10] := B#16#0;
   DP_2.DATA_FIELD[11] := B#16#0;
   DP_2.DATA_FIELD[12] := B#16#0;
   DP_2.DATA_FIELD[13] := B#16#0;
   DP_2.DATA_FIELD[14] := B#16#0;
   DP_2.DATA_FIELD[15] := B#16#0;
   DP_2.DATA_FIELD[16] := B#16#0;
   DP_2.DATA_FIELD[17] := B#16#0;
   DP_2.DATA_FIELD[18] := B#16#0;
   DP_2.DATA_FIELD[19] := B#16#0;
   DP_2.DATA_FIELD[20] := B#16#0;
   DP_2.DATA_FIELD[21] := B#16#0;
   DP_2.DATA_FIELD[22] := B#16#0;
   DP_2.DATA_FIELD[23] := B#16#0;
   DP_2.DATA_FIELD[24] := B#16#0;
   DP_2.DATA_FIELD[25] := B#16#0;
   DP_2.DATA_FIELD[26] := B#16#0;
   DP_2.DATA_FIELD[27] := B#16#0;
   DP_2.DATA_FIELD[28] := B#16#0;
   DP_2.DATA_FIELD[29] := B#16#0;
   DP_2.DATA_FIELD[30] := B#16#0;
   DP_2.DATA_FIELD[31] := B#16#0;
   DP_2.DATA_FIELD[32] := B#16#0;
   DP_2.DATA_FIELD[33] := B#16#0;
   DP_2.DATA_FIELD[34] := B#16#0;
   DP_2.DATA_FIELD[35] := B#16#0;
   DP_2.DATA_FIELD[36] := B#16#0;
   DP_2.DATA_FIELD[37] := B#16#0;
   DP_2.DATA_FIELD[38] := B#16#0;
   DP_2.DATA_FIELD[39] := B#16#0;
   DP_2.DATA_FIELD[40] := B#16#0;
   DP_2.DATA_FIELD[41] := B#16#0;
   DP_2.DATA_FIELD[42] := B#16#0;
   DP_2.DATA_FIELD[43] := B#16#0;
   DP_2.DATA_FIELD[44] := B#16#0;
   DP_2.DATA_FIELD[45] := B#16#0;
   DP_2.DATA_FIELD[46] := B#16#0;
   DP_2.DATA_FIELD[47] := B#16#0;
   DP_2.DATA_FIELD[48] := B#16#0;
   DP_2.DATA_FIELD[49] := B#16#0;
   DP_2.DATA_FIELD[50] := B#16#0;
   DP_2.DATA_FIELD[51] := B#16#0;
   DP_2.DATA_FIELD[52] := B#16#0;
   DP_2.DATA_FIELD[53] := B#16#0;
   DP_2.DATA_FIELD[54] := B#16#0;
   DP_2.SUM_SLAVE_DIAG := 0;
   DP_2.LIST_NOT_PRESENT[0] := DW#16#0;
   DP_2.LIST_NOT_PRESENT[1] := DW#16#0;
   DP_2.LIST_NOT_PRESENT[2] := DW#16#0;
   DP_2.LIST_NOT_PRESENT[3] := DW#16#0;
   DP_2.LIST_ERROR[0] := DW#16#0;
   DP_2.LIST_ERROR[1] := DW#16#0;
   DP_2.LIST_ERROR[2] := DW#16#0;
   DP_2.LIST_ERROR[3] := DW#16#0;
   DP_2.RET_VALUE := 0;
   DP_2.DIAG_EVENT := FALSE;
   DP_2.STATION_ERR := FALSE;
   DP_2.RESTART := FALSE;
   DP_2.BUSY := FALSE;
   DP_2.SP1 := W#16#0;
   DP_2.SP2 := W#16#0;
   DP_3.NDR := FALSE;
   DP_3.ERR := FALSE;
   DP_3.SP21[0] := W#16#0;
   DP_3.SP21[1] := W#16#0;
   DP_3.SP21[2] := W#16#0;
   DP_3.SP21[3] := W#16#0;
   DP_3.STATUS := W#16#8182;
   DP_3.SP22 := W#16#0;
   DP_3.DIAGLNG := B#16#6;
   DP_3.SP23[0] := B#16#0;
   DP_3.SP23[1] := B#16#0;
   DP_3.SP23[2] := B#16#0;
   DP_3.SP23[3] := B#16#0;
   DP_3.LIST_ERROR[0] := DW#16#20000000;
   DP_3.LIST_ERROR[1] := DW#16#0;
   DP_3.LIST_ERROR[2] := DW#16#0;
   DP_3.LIST_ERROR[3] := DW#16#0;
   DP_3.SP24[0] := B#16#0;
   DP_3.SP24[1] := B#16#0;
   DP_3.SP24[2] := B#16#0;
   DP_3.SP24[3] := B#16#0;
   DP_3.SP24[4] := B#16#0;
   DP_3.SP24[5] := B#16#0;
   DP_3.SP24[6] := B#16#0;
   DP_3.SP24[7] := B#16#0;
   DP_3.SP24[8] := B#16#0;
   DP_3.SP24[9] := B#16#0;
   DP_3.SP24[10] := B#16#0;
   DP_3.SP24[11] := B#16#0;
   DP_3.SP24[12] := B#16#0;
   DP_4.NDR := FALSE;
   DP_4.ERR := FALSE;
   DP_4.SP21[0] := W#16#0;
   DP_4.SP21[1] := W#16#0;
   DP_4.SP21[2] := W#16#0;
   DP_4.SP21[3] := W#16#0;
   DP_4.STATUS := W#16#8182;
   DP_4.SP22 := W#16#0;
   DP_4.DIAGLNG := B#16#6;
   DP_4.SP23[0] := B#16#0;
   DP_4.SP23[1] := B#16#0;
   DP_4.SP23[2] := B#16#0;
   DP_4.SP23[3] := B#16#0;
   DP_4.LIST_ERROR[0] := DW#16#20000000;
   DP_4.LIST_ERROR[1] := DW#16#0;
   DP_4.LIST_ERROR[2] := DW#16#0;
   DP_4.LIST_ERROR[3] := DW#16#0;
   DP_4.SP24[0] := B#16#0;
   DP_4.SP24[1] := B#16#0;
   DP_4.SP24[2] := B#16#0;
   DP_4.SP24[3] := B#16#0;
   DP_4.SP24[4] := B#16#0;
   DP_4.SP24[5] := B#16#0;
   DP_4.SP24[6] := B#16#0;
   DP_4.SP24[7] := B#16#0;
   DP_4.SP24[8] := B#16#0;
   DP_4.SP24[9] := B#16#0;
   DP_4.SP24[10] := B#16#0;
   DP_4.SP24[11] := B#16#0;
   DP_4.SP24[12] := B#16#0;
   DP_5.NDR := FALSE;
   DP_5.ERR := FALSE;
   DP_5.SP21[0] := W#16#0;
   DP_5.SP21[1] := W#16#0;
   DP_5.SP21[2] := W#16#0;
   DP_5.SP21[3] := W#16#0;
   DP_5.STATUS := W#16#8182;
   DP_5.SP22 := W#16#0;
   DP_5.DIAGLNG := B#16#6;
   DP_5.SP23[0] := B#16#0;
   DP_5.SP23[1] := B#16#0;
   DP_5.SP23[2] := B#16#0;
   DP_5.SP23[3] := B#16#0;
   DP_5.LIST_ERROR[0] := DW#16#20000000;
   DP_5.LIST_ERROR[1] := DW#16#0;
   DP_5.LIST_ERROR[2] := DW#16#0;
   DP_5.LIST_ERROR[3] := DW#16#0;
   DP_5.SP24[0] := B#16#0;
   DP_5.SP24[1] := B#16#0;
   DP_5.SP24[2] := B#16#0;
   DP_5.SP24[3] := B#16#0;
   DP_5.SP24[4] := B#16#0;
   DP_5.SP24[5] := B#16#0;
   DP_5.SP24[6] := B#16#0;
   DP_5.SP24[7] := B#16#0;
   DP_5.SP24[8] := B#16#0;
   DP_5.SP24[9] := B#16#0;
   DP_5.SP24[10] := B#16#0;
   DP_5.SP24[11] := B#16#0;
   DP_5.SP24[12] := B#16#0;
   DP_6.NDR := FALSE;
   DP_6.ERR := FALSE;
   DP_6.SP21[0] := W#16#0;
   DP_6.SP21[1] := W#16#0;
   DP_6.SP21[2] := W#16#0;
   DP_6.SP21[3] := W#16#0;
   DP_6.STATUS := W#16#8182;
   DP_6.SP22 := W#16#0;
   DP_6.DIAGLNG := B#16#6;
   DP_6.SP23[0] := B#16#0;
   DP_6.SP23[1] := B#16#0;
   DP_6.SP23[2] := B#16#0;
   DP_6.SP23[3] := B#16#0;
   DP_6.LIST_ERROR[0] := DW#16#30000000;
   DP_6.LIST_ERROR[1] := DW#16#0;
   DP_6.LIST_ERROR[2] := DW#16#0;
   DP_6.LIST_ERROR[3] := DW#16#0;
   DP_6.SP24[0] := B#16#0;
   DP_6.SP24[1] := B#16#0;
   DP_6.SP24[2] := B#16#0;
   DP_6.SP24[3] := B#16#0;
   DP_6.SP24[4] := B#16#0;
   DP_6.SP24[5] := B#16#0;
   DP_6.SP24[6] := B#16#0;
   DP_6.SP24[7] := B#16#0;
   DP_6.SP24[8] := B#16#0;
   DP_6.SP24[9] := B#16#0;
   DP_6.SP24[10] := B#16#0;
   DP_6.SP24[11] := B#16#0;
   DP_6.SP24[12] := B#16#0;
   DP_7.NDR := FALSE;
   DP_7.ERR := FALSE;
   DP_7.SP21[0] := W#16#0;
   DP_7.SP21[1] := W#16#0;
   DP_7.SP21[2] := W#16#0;
   DP_7.SP21[3] := W#16#0;
   DP_7.STATUS := W#16#0;
   DP_7.SP22 := W#16#0;
   DP_7.DIAGLNG := B#16#0;
   DP_7.SP23[0] := B#16#0;
   DP_7.SP23[1] := B#16#0;
   DP_7.SP23[2] := B#16#0;
   DP_7.SP23[3] := B#16#0;
   DP_7.LIST_ERROR[0] := DW#16#0;
   DP_7.LIST_ERROR[1] := DW#16#0;
   DP_7.LIST_ERROR[2] := DW#16#0;
   DP_7.LIST_ERROR[3] := DW#16#0;
   DP_7.SP24[0] := B#16#0;
   DP_7.SP24[1] := B#16#0;
   DP_7.SP24[2] := B#16#0;
   DP_7.SP24[3] := B#16#0;
   DP_7.SP24[4] := B#16#0;
   DP_7.SP24[5] := B#16#0;
   DP_7.SP24[6] := B#16#0;
   DP_7.SP24[7] := B#16#0;
   DP_7.SP24[8] := B#16#0;
   DP_7.SP24[9] := B#16#0;
   DP_7.SP24[10] := B#16#0;
   DP_7.SP24[11] := B#16#0;
   DP_7.SP24[12] := B#16#0;
   DP_8.NDR := FALSE;
   DP_8.ERR := FALSE;
   DP_8.SP21[0] := W#16#0;
   DP_8.SP21[1] := W#16#0;
   DP_8.SP21[2] := W#16#0;
   DP_8.SP21[3] := W#16#0;
   DP_8.STATUS := W#16#0;
   DP_8.SP22 := W#16#0;
   DP_8.DIAGLNG := B#16#0;
   DP_8.SP23[0] := B#16#0;
   DP_8.SP23[1] := B#16#0;
   DP_8.SP23[2] := B#16#0;
   DP_8.SP23[3] := B#16#0;
   DP_8.LIST_ERROR[0] := DW#16#0;
   DP_8.LIST_ERROR[1] := DW#16#0;
   DP_8.LIST_ERROR[2] := DW#16#0;
   DP_8.LIST_ERROR[3] := DW#16#0;
   DP_8.SP24[0] := B#16#0;
   DP_8.SP24[1] := B#16#0;
   DP_8.SP24[2] := B#16#0;
   DP_8.SP24[3] := B#16#0;
   DP_8.SP24[4] := B#16#0;
   DP_8.SP24[5] := B#16#0;
   DP_8.SP24[6] := B#16#0;
   DP_8.SP24[7] := B#16#0;
   DP_8.SP24[8] := B#16#0;
   DP_8.SP24[9] := B#16#0;
   DP_8.SP24[10] := B#16#0;
   DP_8.SP24[11] := B#16#0;
   DP_8.SP24[12] := B#16#0;
   DP_9.NDR := FALSE;
   DP_9.ERR := FALSE;
   DP_9.SP21[0] := W#16#0;
   DP_9.SP21[1] := W#16#0;
   DP_9.SP21[2] := W#16#0;
   DP_9.SP21[3] := W#16#0;
   DP_9.STATUS := W#16#0;
   DP_9.SP22 := W#16#0;
   DP_9.DIAGLNG := B#16#0;
   DP_9.SP23[0] := B#16#0;
   DP_9.SP23[1] := B#16#0;
   DP_9.SP23[2] := B#16#0;
   DP_9.SP23[3] := B#16#0;
   DP_9.LIST_ERROR[0] := DW#16#0;
   DP_9.LIST_ERROR[1] := DW#16#0;
   DP_9.LIST_ERROR[2] := DW#16#0;
   DP_9.LIST_ERROR[3] := DW#16#0;
   DP_9.SP24[0] := B#16#0;
   DP_9.SP24[1] := B#16#0;
   DP_9.SP24[2] := B#16#0;
   DP_9.SP24[3] := B#16#0;
   DP_9.SP24[4] := B#16#0;
   DP_9.SP24[5] := B#16#0;
   DP_9.SP24[6] := B#16#0;
   DP_9.SP24[7] := B#16#0;
   DP_9.SP24[8] := B#16#0;
   DP_9.SP24[9] := B#16#0;
   DP_9.SP24[10] := B#16#0;
   DP_9.SP24[11] := B#16#0;
   DP_9.SP24[12] := B#16#0;
   DP_10.NDR := FALSE;
   DP_10.ERR := FALSE;
   DP_10.SP21[0] := W#16#0;
   DP_10.SP21[1] := W#16#0;
   DP_10.SP21[2] := W#16#0;
   DP_10.SP21[3] := W#16#0;
   DP_10.STATUS := W#16#0;
   DP_10.SP22 := W#16#0;
   DP_10.DIAGLNG := B#16#0;
   DP_10.SP23[0] := B#16#0;
   DP_10.SP23[1] := B#16#0;
   DP_10.SP23[2] := B#16#0;
   DP_10.SP23[3] := B#16#0;
   DP_10.LIST_ERROR[0] := DW#16#0;
   DP_10.LIST_ERROR[1] := DW#16#0;
   DP_10.LIST_ERROR[2] := DW#16#0;
   DP_10.LIST_ERROR[3] := DW#16#0;
   DP_10.SP24[0] := B#16#0;
   DP_10.SP24[1] := B#16#0;
   DP_10.SP24[2] := B#16#0;
   DP_10.SP24[3] := B#16#0;
   DP_10.SP24[4] := B#16#0;
   DP_10.SP24[5] := B#16#0;
   DP_10.SP24[6] := B#16#0;
   DP_10.SP24[7] := B#16#0;
   DP_10.SP24[8] := B#16#0;
   DP_10.SP24[9] := B#16#0;
   DP_10.SP24[10] := B#16#0;
   DP_10.SP24[11] := B#16#0;
   DP_10.SP24[12] := B#16#0;
END_DATA_BLOCK

DATA_BLOCK DB 55
TITLE =
VERSION : 0.1


  STRUCT
   CP1 : STRUCT
    FC2_NDR : BOOL ;
    FC2_ERROR : BOOL ;
    SP1 : BOOL ;
    SP2 : BOOL ;
    FC1_NDR : BOOL ;
    FC1_ERROR : BOOL ;
    SP3 : BOOL ;
    SP4 : BOOL ;
    FC2_STATUS : WORD ;
    FC2_DPSTATUS : BYTE ;
    FC1_STATUS : WORD ;
    SP5 : WORD ;
    SFC20_1_RET_VAL : INT ;
    SFC20_2_RET_VAL : INT ;
    SFC20_3_RET_VAL : INT ;
    SFC20_4_RET_VAL : INT ;
    SFC20_5_RET_VAL : INT ;
    SFC20_6_RET_VAL : INT ;
    SFC20_7_RET_VAL : INT ;
    SFC20_8_RET_VAL : INT ;
    SFC20_9_RET_VAL : INT ;
    SFC20_10_RET_VAL : INT ;
    SP : ARRAY  [0 .. 9 ] OF WORD ;
   END_STRUCT ;
   CP2 : STRUCT
    FC2_NDR : BOOL ;
    FC2_ERROR : BOOL ;
    SP1 : BOOL ;
    SP2 : BOOL ;
    FC1_NDR : BOOL ;
    FC1_ERROR : BOOL ;
    SP3 : BOOL ;
    SP4 : BOOL ;
    FC2_STATUS : WORD ;
    FC2_DPSTATUS : BYTE ;
    FC1_STATUS : WORD ;
    SP5 : WORD ;
    SFC20_1_RET_VAL : INT ;
    SFC20_2_RET_VAL : INT ;
    SFC20_3_RET_VAL : INT ;
    SFC20_4_RET_VAL : INT ;
    SFC20_5_RET_VAL : INT ;
    SFC20_6_RET_VAL : INT ;
    SFC20_7_RET_VAL : INT ;
    SFC20_8_RET_VAL : INT ;
    SFC20_9_RET_VAL : INT ;
    SFC20_10_RET_VAL : INT ;
    SP : ARRAY  [0 .. 9 ] OF WORD ;
   END_STRUCT ;
   CP3 : STRUCT
    FC2_NDR : BOOL ;
    FC2_ERROR : BOOL ;
    SP1 : BOOL ;
    SP2 : BOOL ;
    FC1_NDR : BOOL ;
    FC1_ERROR : BOOL ;
    SP3 : BOOL ;
    SP4 : BOOL ;
    FC2_STATUS : WORD ;
    FC2_DPSTATUS : BYTE ;
    FC1_STATUS : WORD ;
    SP5 : WORD ;
    SFC20_1_RET_VAL : INT ;
    SFC20_2_RET_VAL : INT ;
    SFC20_3_RET_VAL : INT ;
    SFC20_4_RET_VAL : INT ;
    SFC20_5_RET_VAL : INT ;
    SFC20_6_RET_VAL : INT ;
    SFC20_7_RET_VAL : INT ;
    SFC20_8_RET_VAL : INT ;
    SFC20_9_RET_VAL : INT ;
    SFC20_10_RET_VAL : INT ;
    SP : ARRAY  [0 .. 9 ] OF WORD ;
   END_STRUCT ;
   CP4 : STRUCT
    FC2_NDR : BOOL ;
    FC2_ERROR : BOOL ;
    SP1 : BOOL ;
    SP2 : BOOL ;
    FC1_NDR : BOOL ;
    FC1_ERROR : BOOL ;
    SP3 : BOOL ;
    SP4 : BOOL ;
    FC2_STATUS : WORD ;
    FC2_DPSTATUS : BYTE ;
    FC1_STATUS : WORD ;
    SP5 : WORD ;
    SFC20_1_RET_VAL : INT ;
    SFC20_2_RET_VAL : INT ;
    SFC20_3_RET_VAL : INT ;
    SFC20_4_RET_VAL : INT ;
    SFC20_5_RET_VAL : INT ;
    SFC20_6_RET_VAL : INT ;
    SFC20_7_RET_VAL : INT ;
    SFC20_8_RET_VAL : INT ;
    SFC20_9_RET_VAL : INT ;
    SFC20_10_RET_VAL : INT ;
    SP : ARRAY  [0 .. 9 ] OF WORD ;
   END_STRUCT ;
   CP5 : STRUCT
    FC2_NDR : BOOL ;
    FC2_ERROR : BOOL ;
    SP1 : BOOL ;
    SP2 : BOOL ;
    FC1_NDR : BOOL ;
    FC1_ERROR : BOOL ;
    SP3 : BOOL ;
    SP4 : BOOL ;
    FC2_STATUS : WORD ;
    FC2_DPSTATUS : BYTE ;
    FC1_STATUS : WORD ;
    SP5 : WORD ;
    SFC20_1_RET_VAL : INT ;
    SFC20_2_RET_VAL : INT ;
    SFC20_3_RET_VAL : INT ;
    SFC20_4_RET_VAL : INT ;
    SFC20_5_RET_VAL : INT ;
    SFC20_6_RET_VAL : INT ;
    SFC20_7_RET_VAL : INT ;
    SFC20_8_RET_VAL : INT ;
    SFC20_9_RET_VAL : INT ;
    SFC20_10_RET_VAL : INT ;
    SP : ARRAY  [0 .. 9 ] OF WORD ;
   END_STRUCT ;
   CP6 : STRUCT
    FC2_NDR : BOOL ;
    FC2_ERROR : BOOL ;
    SP1 : BOOL ;
    SP2 : BOOL ;
    FC1_NDR : BOOL ;
    FC1_ERROR : BOOL ;
    SP3 : BOOL ;
    SP4 : BOOL ;
    FC2_STATUS : WORD ;
    FC2_DPSTATUS : BYTE ;
    FC1_STATUS : WORD ;
    SP5 : WORD ;
    SFC20_1_RET_VAL : INT ;
    SFC20_2_RET_VAL : INT ;
    SFC20_3_RET_VAL : INT ;
    SFC20_4_RET_VAL : INT ;
    SFC20_5_RET_VAL : INT ;
    SFC20_6_RET_VAL : INT ;
    SFC20_7_RET_VAL : INT ;
    SFC20_8_RET_VAL : INT ;
    SFC20_9_RET_VAL : INT ;
    SFC20_10_RET_VAL : INT ;
    SP : ARRAY  [0 .. 9 ] OF WORD ;
   END_STRUCT ;
   CP7 : STRUCT
    FC2_NDR : BOOL ;
    FC2_ERROR : BOOL ;
    SP1 : BOOL ;
    SP2 : BOOL ;
    FC1_NDR : BOOL ;
    FC1_ERROR : BOOL ;
    SP3 : BOOL ;
    SP4 : BOOL ;
    FC2_STATUS : WORD ;
    FC2_DPSTATUS : BYTE ;
    FC1_STATUS : WORD ;
    SP5 : WORD ;
    SFC20_1_RET_VAL : INT ;
    SFC20_2_RET_VAL : INT ;
    SFC20_3_RET_VAL : INT ;
    SFC20_4_RET_VAL : INT ;
    SFC20_5_RET_VAL : INT ;
    SFC20_6_RET_VAL : INT ;
    SFC20_7_RET_VAL : INT ;
    SFC20_8_RET_VAL : INT ;
    SFC20_9_RET_VAL : INT ;
    SFC20_10_RET_VAL : INT ;
    SP : ARRAY  [0 .. 9 ] OF WORD ;
   END_STRUCT ;
   CP8 : STRUCT
    FC2_NDR : BOOL ;
    FC2_ERROR : BOOL ;
    SP1 : BOOL ;
    SP2 : BOOL ;
    FC1_NDR : BOOL ;
    FC1_ERROR : BOOL ;
    SP3 : BOOL ;
    SP4 : BOOL ;
    FC2_STATUS : WORD ;
    FC2_DPSTATUS : BYTE ;
    FC1_STATUS : WORD ;
    SP5 : WORD ;
    SFC20_1_RET_VAL : INT ;
    SFC20_2_RET_VAL : INT ;
    SFC20_3_RET_VAL : INT ;
    SFC20_4_RET_VAL : INT ;
    SFC20_5_RET_VAL : INT ;
    SFC20_6_RET_VAL : INT ;
    SFC20_7_RET_VAL : INT ;
    SFC20_8_RET_VAL : INT ;
    SFC20_9_RET_VAL : INT ;
    SFC20_10_RET_VAL : INT ;
    SP : ARRAY  [0 .. 9 ] OF WORD ;
   END_STRUCT ;
   RTN_VALUE_WORD : ARRAY  [0 .. 49 ] OF WORD ;
   AG1 : STRUCT
    FC6_NDR : BOOL ;
    FC6_ERROR : BOOL ;
    SP1 : BOOL ;
    SP2 : BOOL ;
    FC5_NDR : BOOL ;
    FC5_ERROR : BOOL ;
    SP3 : BOOL ;
    SP4 : BOOL ;
    FC6_STATUS : WORD ;
    FC6_DPSTATUS : BYTE ;
    FC5_STATUS : WORD ;
    SP5 : WORD ;
    SFC20_1_RET_VAL : INT ;
    SFC20_2_RET_VAL : INT ;
    SFC20_3_RET_VAL : INT ;
    SFC20_4_RET_VAL : INT ;
    SFC20_5_RET_VAL : INT ;
    SFC20_6_RET_VAL : INT ;
    SFC20_7_RET_VAL : INT ;
    SFC20_8_RET_VAL : INT ;
    SFC20_9_RET_VAL : INT ;
    SFC20_10_RET_VAL : INT ;
    SP : ARRAY  [0 .. 9 ] OF WORD ;
   END_STRUCT ;
   AG2 : STRUCT
    FC6_NDR : BOOL ;
    FC6_ERROR : BOOL ;
    SP1 : BOOL ;
    SP2 : BOOL ;
    FC5_NDR : BOOL ;
    FC5_ERROR : BOOL ;
    SP3 : BOOL ;
    SP4 : BOOL ;
    FC6_STATUS : WORD ;
    FC6_DPSTATUS : BYTE ;
    FC5_STATUS : WORD ;
    SP5 : WORD ;
    SFC20_1_RET_VAL : INT ;
    SFC20_2_RET_VAL : INT ;
    SFC20_3_RET_VAL : INT ;
    SFC20_4_RET_VAL : INT ;
    SFC20_5_RET_VAL : INT ;
    SFC20_6_RET_VAL : INT ;
    SFC20_7_RET_VAL : INT ;
    SFC20_8_RET_VAL : INT ;
    SFC20_9_RET_VAL : INT ;
    SFC20_10_RET_VAL : INT ;
    SP : ARRAY  [0 .. 9 ] OF WORD ;
   END_STRUCT ;
   AG3 : STRUCT
    FC6_NDR : BOOL ;
    FC6_ERROR : BOOL ;
    SP1 : BOOL ;
    SP2 : BOOL ;
    FC5_NDR : BOOL ;
    FC5_ERROR : BOOL ;
    SP3 : BOOL ;
    SP4 : BOOL ;
    FC6_STATUS : WORD ;
    FC6_DPSTATUS : BYTE ;
    FC5_STATUS : WORD ;
    SP5 : WORD ;
    SFC20_1_RET_VAL : INT ;
    SFC20_2_RET_VAL : INT ;
    SFC20_3_RET_VAL : INT ;
    SFC20_4_RET_VAL : INT ;
    SFC20_5_RET_VAL : INT ;
    SFC20_6_RET_VAL : INT ;
    SFC20_7_RET_VAL : INT ;
    SFC20_8_RET_VAL : INT ;
    SFC20_9_RET_VAL : INT ;
    SFC20_10_RET_VAL : INT ;
    SP : ARRAY  [0 .. 9 ] OF WORD ;
   END_STRUCT ;
   AG4 : STRUCT
    FC6_NDR : BOOL ;
    FC6_ERROR : BOOL ;
    SP1 : BOOL ;
    SP2 : BOOL ;
    FC5_NDR : BOOL ;
    FC5_ERROR : BOOL ;
    SP3 : BOOL ;
    SP4 : BOOL ;
    FC6_STATUS : WORD ;
    FC6_DPSTATUS : BYTE ;
    FC5_STATUS : WORD ;
    SP5 : WORD ;
    SFC20_1_RET_VAL : INT ;
    SFC20_2_RET_VAL : INT ;
    SFC20_3_RET_VAL : INT ;
    SFC20_4_RET_VAL : INT ;
    SFC20_5_RET_VAL : INT ;
    SFC20_6_RET_VAL : INT ;
    SFC20_7_RET_VAL : INT ;
    SFC20_8_RET_VAL : INT ;
    SFC20_9_RET_VAL : INT ;
    SFC20_10_RET_VAL : INT ;
    SP : ARRAY  [0 .. 9 ] OF WORD ;
   END_STRUCT ;
   AG5 : STRUCT
    FC6_NDR : BOOL ;
    FC6_ERROR : BOOL ;
    SP1 : BOOL ;
    SP2 : BOOL ;
    FC5_NDR : BOOL ;
    FC5_ERROR : BOOL ;
    SP3 : BOOL ;
    SP4 : BOOL ;
    FC6_STATUS : WORD ;
    FC6_DPSTATUS : BYTE ;
    FC5_STATUS : WORD ;
    SP5 : WORD ;
    SFC20_1_RET_VAL : INT ;
    SFC20_2_RET_VAL : INT ;
    SFC20_3_RET_VAL : INT ;
    SFC20_4_RET_VAL : INT ;
    SFC20_5_RET_VAL : INT ;
    SFC20_6_RET_VAL : INT ;
    SFC20_7_RET_VAL : INT ;
    SFC20_8_RET_VAL : INT ;
    SFC20_9_RET_VAL : INT ;
    SFC20_10_RET_VAL : INT ;
    SP : ARRAY  [0 .. 9 ] OF WORD ;
   END_STRUCT ;
   AG6 : STRUCT
    FC6_NDR : BOOL ;
    FC6_ERROR : BOOL ;
    SP1 : BOOL ;
    SP2 : BOOL ;
    FC5_NDR : BOOL ;
    FC5_ERROR : BOOL ;
    SP3 : BOOL ;
    SP4 : BOOL ;
    FC6_STATUS : WORD ;
    FC6_DPSTATUS : BYTE ;
    FC5_STATUS : WORD ;
    SP5 : WORD ;
    SFC20_1_RET_VAL : INT ;
    SFC20_2_RET_VAL : INT ;
    SFC20_3_RET_VAL : INT ;
    SFC20_4_RET_VAL : INT ;
    SFC20_5_RET_VAL : INT ;
    SFC20_6_RET_VAL : INT ;
    SFC20_7_RET_VAL : INT ;
    SFC20_8_RET_VAL : INT ;
    SFC20_9_RET_VAL : INT ;
    SFC20_10_RET_VAL : INT ;
    SP : ARRAY  [0 .. 9 ] OF WORD ;
   END_STRUCT ;
   AG7 : STRUCT
    FC6_NDR : BOOL ;
    FC6_ERROR : BOOL ;
    SP1 : BOOL ;
    SP2 : BOOL ;
    FC5_NDR : BOOL ;
    FC5_ERROR : BOOL ;
    SP3 : BOOL ;
    SP4 : BOOL ;
    FC6_STATUS : WORD ;
    FC6_DPSTATUS : BYTE ;
    FC5_STATUS : WORD ;
    SP5 : WORD ;
    SFC20_1_RET_VAL : INT ;
    SFC20_2_RET_VAL : INT ;
    SFC20_3_RET_VAL : INT ;
    SFC20_4_RET_VAL : INT ;
    SFC20_5_RET_VAL : INT ;
    SFC20_6_RET_VAL : INT ;
    SFC20_7_RET_VAL : INT ;
    SFC20_8_RET_VAL : INT ;
    SFC20_9_RET_VAL : INT ;
    SFC20_10_RET_VAL : INT ;
    SP : ARRAY  [0 .. 9 ] OF WORD ;
   END_STRUCT ;
   SP : ARRAY  [0 .. 74 ] OF WORD ;
   CTYPE_RET_VAL : ARRAY  [0 .. 99 ] OF INT ;
   MES_RET_VAL1 : ARRAY  [0 .. 199 ] OF INT ;
  END_STRUCT ;
BEGIN
   CP1.FC2_NDR := TRUE;
   CP1.FC2_ERROR := FALSE;
   CP1.SP1 := FALSE;
   CP1.SP2 := FALSE;
   CP1.FC1_NDR := FALSE;
   CP1.FC1_ERROR := FALSE;
   CP1.SP3 := FALSE;
   CP1.SP4 := FALSE;
   CP1.FC2_STATUS := W#16#0;
   CP1.FC2_DPSTATUS := B#16#6;
   CP1.FC1_STATUS := W#16#8180;
   CP1.SP5 := W#16#0;
   CP1.SFC20_1_RET_VAL := 0;
   CP1.SFC20_2_RET_VAL := 0;
   CP1.SFC20_3_RET_VAL := 0;
   CP1.SFC20_4_RET_VAL := 0;
   CP1.SFC20_5_RET_VAL := 0;
   CP1.SFC20_6_RET_VAL := 0;
   CP1.SFC20_7_RET_VAL := 0;
   CP1.SFC20_8_RET_VAL := 0;
   CP1.SFC20_9_RET_VAL := 0;
   CP1.SFC20_10_RET_VAL := 0;
   CP1.SP[0] := W#16#0;
   CP1.SP[1] := W#16#0;
   CP1.SP[2] := W#16#0;
   CP1.SP[3] := W#16#0;
   CP1.SP[4] := W#16#0;
   CP1.SP[5] := W#16#0;
   CP1.SP[6] := W#16#0;
   CP1.SP[7] := W#16#0;
   CP1.SP[8] := W#16#0;
   CP1.SP[9] := W#16#0;
   CP2.FC2_NDR := TRUE;
   CP2.FC2_ERROR := FALSE;
   CP2.SP1 := FALSE;
   CP2.SP2 := FALSE;
   CP2.FC1_NDR := FALSE;
   CP2.FC1_ERROR := FALSE;
   CP2.SP3 := FALSE;
   CP2.SP4 := FALSE;
   CP2.FC2_STATUS := W#16#0;
   CP2.FC2_DPSTATUS := B#16#6;
   CP2.FC1_STATUS := W#16#8180;
   CP2.SP5 := W#16#0;
   CP2.SFC20_1_RET_VAL := 0;
   CP2.SFC20_2_RET_VAL := 0;
   CP2.SFC20_3_RET_VAL := 0;
   CP2.SFC20_4_RET_VAL := 0;
   CP2.SFC20_5_RET_VAL := 0;
   CP2.SFC20_6_RET_VAL := 0;
   CP2.SFC20_7_RET_VAL := 0;
   CP2.SFC20_8_RET_VAL := 0;
   CP2.SFC20_9_RET_VAL := 0;
   CP2.SFC20_10_RET_VAL := 0;
   CP2.SP[0] := W#16#0;
   CP2.SP[1] := W#16#0;
   CP2.SP[2] := W#16#0;
   CP2.SP[3] := W#16#0;
   CP2.SP[4] := W#16#0;
   CP2.SP[5] := W#16#0;
   CP2.SP[6] := W#16#0;
   CP2.SP[7] := W#16#0;
   CP2.SP[8] := W#16#0;
   CP2.SP[9] := W#16#0;
   CP3.FC2_NDR := TRUE;
   CP3.FC2_ERROR := FALSE;
   CP3.SP1 := FALSE;
   CP3.SP2 := FALSE;
   CP3.FC1_NDR := FALSE;
   CP3.FC1_ERROR := FALSE;
   CP3.SP3 := FALSE;
   CP3.SP4 := FALSE;
   CP3.FC2_STATUS := W#16#0;
   CP3.FC2_DPSTATUS := B#16#6;
   CP3.FC1_STATUS := W#16#8180;
   CP3.SP5 := W#16#0;
   CP3.SFC20_1_RET_VAL := 0;
   CP3.SFC20_2_RET_VAL := 0;
   CP3.SFC20_3_RET_VAL := 0;
   CP3.SFC20_4_RET_VAL := 0;
   CP3.SFC20_5_RET_VAL := 0;
   CP3.SFC20_6_RET_VAL := 0;
   CP3.SFC20_7_RET_VAL := 0;
   CP3.SFC20_8_RET_VAL := 0;
   CP3.SFC20_9_RET_VAL := 0;
   CP3.SFC20_10_RET_VAL := 0;
   CP3.SP[0] := W#16#0;
   CP3.SP[1] := W#16#0;
   CP3.SP[2] := W#16#0;
   CP3.SP[3] := W#16#0;
   CP3.SP[4] := W#16#0;
   CP3.SP[5] := W#16#0;
   CP3.SP[6] := W#16#0;
   CP3.SP[7] := W#16#0;
   CP3.SP[8] := W#16#0;
   CP3.SP[9] := W#16#0;
   CP4.FC2_NDR := TRUE;
   CP4.FC2_ERROR := FALSE;
   CP4.SP1 := FALSE;
   CP4.SP2 := FALSE;
   CP4.FC1_NDR := FALSE;
   CP4.FC1_ERROR := FALSE;
   CP4.SP3 := FALSE;
   CP4.SP4 := FALSE;
   CP4.FC2_STATUS := W#16#0;
   CP4.FC2_DPSTATUS := B#16#6;
   CP4.FC1_STATUS := W#16#8180;
   CP4.SP5 := W#16#0;
   CP4.SFC20_1_RET_VAL := 0;
   CP4.SFC20_2_RET_VAL := 0;
   CP4.SFC20_3_RET_VAL := 0;
   CP4.SFC20_4_RET_VAL := 0;
   CP4.SFC20_5_RET_VAL := 0;
   CP4.SFC20_6_RET_VAL := 0;
   CP4.SFC20_7_RET_VAL := 0;
   CP4.SFC20_8_RET_VAL := 0;
   CP4.SFC20_9_RET_VAL := 0;
   CP4.SFC20_10_RET_VAL := 0;
   CP4.SP[0] := W#16#0;
   CP4.SP[1] := W#16#0;
   CP4.SP[2] := W#16#0;
   CP4.SP[3] := W#16#0;
   CP4.SP[4] := W#16#0;
   CP4.SP[5] := W#16#0;
   CP4.SP[6] := W#16#0;
   CP4.SP[7] := W#16#0;
   CP4.SP[8] := W#16#0;
   CP4.SP[9] := W#16#0;
   CP5.FC2_NDR := FALSE;
   CP5.FC2_ERROR := FALSE;
   CP5.SP1 := FALSE;
   CP5.SP2 := FALSE;
   CP5.FC1_NDR := FALSE;
   CP5.FC1_ERROR := FALSE;
   CP5.SP3 := FALSE;
   CP5.SP4 := FALSE;
   CP5.FC2_STATUS := W#16#8180;
   CP5.FC2_DPSTATUS := B#16#0;
   CP5.FC1_STATUS := W#16#8180;
   CP5.SP5 := W#16#0;
   CP5.SFC20_1_RET_VAL := 0;
   CP5.SFC20_2_RET_VAL := 0;
   CP5.SFC20_3_RET_VAL := 0;
   CP5.SFC20_4_RET_VAL := 0;
   CP5.SFC20_5_RET_VAL := 0;
   CP5.SFC20_6_RET_VAL := 0;
   CP5.SFC20_7_RET_VAL := 0;
   CP5.SFC20_8_RET_VAL := 0;
   CP5.SFC20_9_RET_VAL := 0;
   CP5.SFC20_10_RET_VAL := 0;
   CP5.SP[0] := W#16#0;
   CP5.SP[1] := W#16#0;
   CP5.SP[2] := W#16#0;
   CP5.SP[3] := W#16#0;
   CP5.SP[4] := W#16#0;
   CP5.SP[5] := W#16#0;
   CP5.SP[6] := W#16#0;
   CP5.SP[7] := W#16#0;
   CP5.SP[8] := W#16#0;
   CP5.SP[9] := W#16#0;
   CP6.FC2_NDR := FALSE;
   CP6.FC2_ERROR := FALSE;
   CP6.SP1 := FALSE;
   CP6.SP2 := FALSE;
   CP6.FC1_NDR := FALSE;
   CP6.FC1_ERROR := FALSE;
   CP6.SP3 := FALSE;
   CP6.SP4 := FALSE;
   CP6.FC2_STATUS := W#16#0;
   CP6.FC2_DPSTATUS := B#16#0;
   CP6.FC1_STATUS := W#16#0;
   CP6.SP5 := W#16#0;
   CP6.SFC20_1_RET_VAL := 0;
   CP6.SFC20_2_RET_VAL := 0;
   CP6.SFC20_3_RET_VAL := 0;
   CP6.SFC20_4_RET_VAL := 0;
   CP6.SFC20_5_RET_VAL := 0;
   CP6.SFC20_6_RET_VAL := 0;
   CP6.SFC20_7_RET_VAL := 0;
   CP6.SFC20_8_RET_VAL := 0;
   CP6.SFC20_9_RET_VAL := 0;
   CP6.SFC20_10_RET_VAL := 0;
   CP6.SP[0] := W#16#0;
   CP6.SP[1] := W#16#0;
   CP6.SP[2] := W#16#0;
   CP6.SP[3] := W#16#0;
   CP6.SP[4] := W#16#0;
   CP6.SP[5] := W#16#0;
   CP6.SP[6] := W#16#0;
   CP6.SP[7] := W#16#0;
   CP6.SP[8] := W#16#0;
   CP6.SP[9] := W#16#0;
   CP7.FC2_NDR := FALSE;
   CP7.FC2_ERROR := FALSE;
   CP7.SP1 := FALSE;
   CP7.SP2 := FALSE;
   CP7.FC1_NDR := FALSE;
   CP7.FC1_ERROR := FALSE;
   CP7.SP3 := FALSE;
   CP7.SP4 := FALSE;
   CP7.FC2_STATUS := W#16#0;
   CP7.FC2_DPSTATUS := B#16#0;
   CP7.FC1_STATUS := W#16#0;
   CP7.SP5 := W#16#0;
   CP7.SFC20_1_RET_VAL := 0;
   CP7.SFC20_2_RET_VAL := 0;
   CP7.SFC20_3_RET_VAL := 0;
   CP7.SFC20_4_RET_VAL := 0;
   CP7.SFC20_5_RET_VAL := 0;
   CP7.SFC20_6_RET_VAL := 0;
   CP7.SFC20_7_RET_VAL := 0;
   CP7.SFC20_8_RET_VAL := 0;
   CP7.SFC20_9_RET_VAL := 0;
   CP7.SFC20_10_RET_VAL := 0;
   CP7.SP[0] := W#16#0;
   CP7.SP[1] := W#16#0;
   CP7.SP[2] := W#16#0;
   CP7.SP[3] := W#16#0;
   CP7.SP[4] := W#16#0;
   CP7.SP[5] := W#16#0;
   CP7.SP[6] := W#16#0;
   CP7.SP[7] := W#16#0;
   CP7.SP[8] := W#16#0;
   CP7.SP[9] := W#16#0;
   CP8.FC2_NDR := FALSE;
   CP8.FC2_ERROR := FALSE;
   CP8.SP1 := FALSE;
   CP8.SP2 := FALSE;
   CP8.FC1_NDR := FALSE;
   CP8.FC1_ERROR := FALSE;
   CP8.SP3 := FALSE;
   CP8.SP4 := FALSE;
   CP8.FC2_STATUS := W#16#0;
   CP8.FC2_DPSTATUS := B#16#0;
   CP8.FC1_STATUS := W#16#0;
   CP8.SP5 := W#16#0;
   CP8.SFC20_1_RET_VAL := 0;
   CP8.SFC20_2_RET_VAL := 0;
   CP8.SFC20_3_RET_VAL := 0;
   CP8.SFC20_4_RET_VAL := 0;
   CP8.SFC20_5_RET_VAL := 0;
   CP8.SFC20_6_RET_VAL := 0;
   CP8.SFC20_7_RET_VAL := 0;
   CP8.SFC20_8_RET_VAL := 0;
   CP8.SFC20_9_RET_VAL := 0;
   CP8.SFC20_10_RET_VAL := 0;
   CP8.SP[0] := W#16#0;
   CP8.SP[1] := W#16#0;
   CP8.SP[2] := W#16#0;
   CP8.SP[3] := W#16#0;
   CP8.SP[4] := W#16#0;
   CP8.SP[5] := W#16#0;
   CP8.SP[6] := W#16#0;
   CP8.SP[7] := W#16#0;
   CP8.SP[8] := W#16#0;
   CP8.SP[9] := W#16#0;
   RTN_VALUE_WORD[0] := W#16#0;
   RTN_VALUE_WORD[1] := W#16#0;
   RTN_VALUE_WORD[2] := W#16#0;
   RTN_VALUE_WORD[3] := W#16#0;
   RTN_VALUE_WORD[4] := W#16#0;
   RTN_VALUE_WORD[5] := W#16#0;
   RTN_VALUE_WORD[6] := W#16#0;
   RTN_VALUE_WORD[7] := W#16#0;
   RTN_VALUE_WORD[8] := W#16#0;
   RTN_VALUE_WORD[9] := W#16#0;
   RTN_VALUE_WORD[10] := W#16#0;
   RTN_VALUE_WORD[11] := W#16#0;
   RTN_VALUE_WORD[12] := W#16#0;
   RTN_VALUE_WORD[13] := W#16#0;
   RTN_VALUE_WORD[14] := W#16#0;
   RTN_VALUE_WORD[15] := W#16#0;
   RTN_VALUE_WORD[16] := W#16#0;
   RTN_VALUE_WORD[17] := W#16#0;
   RTN_VALUE_WORD[18] := W#16#0;
   RTN_VALUE_WORD[19] := W#16#0;
   RTN_VALUE_WORD[20] := W#16#0;
   RTN_VALUE_WORD[21] := W#16#0;
   RTN_VALUE_WORD[22] := W#16#0;
   RTN_VALUE_WORD[23] := W#16#0;
   RTN_VALUE_WORD[24] := W#16#0;
   RTN_VALUE_WORD[25] := W#16#0;
   RTN_VALUE_WORD[26] := W#16#0;
   RTN_VALUE_WORD[27] := W#16#0;
   RTN_VALUE_WORD[28] := W#16#0;
   RTN_VALUE_WORD[29] := W#16#0;
   RTN_VALUE_WORD[30] := W#16#0;
   RTN_VALUE_WORD[31] := W#16#0;
   RTN_VALUE_WORD[32] := W#16#0;
   RTN_VALUE_WORD[33] := W#16#0;
   RTN_VALUE_WORD[34] := W#16#0;
   RTN_VALUE_WORD[35] := W#16#0;
   RTN_VALUE_WORD[36] := W#16#0;
   RTN_VALUE_WORD[37] := W#16#0;
   RTN_VALUE_WORD[38] := W#16#0;
   RTN_VALUE_WORD[39] := W#16#0;
   RTN_VALUE_WORD[40] := W#16#0;
   RTN_VALUE_WORD[41] := W#16#0;
   RTN_VALUE_WORD[42] := W#16#0;
   RTN_VALUE_WORD[43] := W#16#0;
   RTN_VALUE_WORD[44] := W#16#0;
   RTN_VALUE_WORD[45] := W#16#0;
   RTN_VALUE_WORD[46] := W#16#0;
   RTN_VALUE_WORD[47] := W#16#0;
   RTN_VALUE_WORD[48] := W#16#0;
   RTN_VALUE_WORD[49] := W#16#0;
   AG1.FC6_NDR := FALSE;
   AG1.FC6_ERROR := FALSE;
   AG1.SP1 := FALSE;
   AG1.SP2 := FALSE;
   AG1.FC5_NDR := FALSE;
   AG1.FC5_ERROR := FALSE;
   AG1.SP3 := FALSE;
   AG1.SP4 := FALSE;
   AG1.FC6_STATUS := W#16#0;
   AG1.FC6_DPSTATUS := B#16#0;
   AG1.FC5_STATUS := W#16#0;
   AG1.SP5 := W#16#0;
   AG1.SFC20_1_RET_VAL := 0;
   AG1.SFC20_2_RET_VAL := 0;
   AG1.SFC20_3_RET_VAL := 0;
   AG1.SFC20_4_RET_VAL := 0;
   AG1.SFC20_5_RET_VAL := 0;
   AG1.SFC20_6_RET_VAL := 0;
   AG1.SFC20_7_RET_VAL := 0;
   AG1.SFC20_8_RET_VAL := 0;
   AG1.SFC20_9_RET_VAL := 0;
   AG1.SFC20_10_RET_VAL := 0;
   AG1.SP[0] := W#16#0;
   AG1.SP[1] := W#16#0;
   AG1.SP[2] := W#16#0;
   AG1.SP[3] := W#16#0;
   AG1.SP[4] := W#16#0;
   AG1.SP[5] := W#16#0;
   AG1.SP[6] := W#16#0;
   AG1.SP[7] := W#16#0;
   AG1.SP[8] := W#16#0;
   AG1.SP[9] := W#16#0;
   AG2.FC6_NDR := FALSE;
   AG2.FC6_ERROR := FALSE;
   AG2.SP1 := FALSE;
   AG2.SP2 := FALSE;
   AG2.FC5_NDR := FALSE;
   AG2.FC5_ERROR := FALSE;
   AG2.SP3 := FALSE;
   AG2.SP4 := FALSE;
   AG2.FC6_STATUS := W#16#0;
   AG2.FC6_DPSTATUS := B#16#0;
   AG2.FC5_STATUS := W#16#0;
   AG2.SP5 := W#16#0;
   AG2.SFC20_1_RET_VAL := 0;
   AG2.SFC20_2_RET_VAL := 0;
   AG2.SFC20_3_RET_VAL := 0;
   AG2.SFC20_4_RET_VAL := 0;
   AG2.SFC20_5_RET_VAL := 0;
   AG2.SFC20_6_RET_VAL := 0;
   AG2.SFC20_7_RET_VAL := 0;
   AG2.SFC20_8_RET_VAL := 0;
   AG2.SFC20_9_RET_VAL := 0;
   AG2.SFC20_10_RET_VAL := 0;
   AG2.SP[0] := W#16#0;
   AG2.SP[1] := W#16#0;
   AG2.SP[2] := W#16#0;
   AG2.SP[3] := W#16#0;
   AG2.SP[4] := W#16#0;
   AG2.SP[5] := W#16#0;
   AG2.SP[6] := W#16#0;
   AG2.SP[7] := W#16#0;
   AG2.SP[8] := W#16#0;
   AG2.SP[9] := W#16#0;
   AG3.FC6_NDR := FALSE;
   AG3.FC6_ERROR := FALSE;
   AG3.SP1 := FALSE;
   AG3.SP2 := FALSE;
   AG3.FC5_NDR := FALSE;
   AG3.FC5_ERROR := FALSE;
   AG3.SP3 := FALSE;
   AG3.SP4 := FALSE;
   AG3.FC6_STATUS := W#16#0;
   AG3.FC6_DPSTATUS := B#16#0;
   AG3.FC5_STATUS := W#16#0;
   AG3.SP5 := W#16#0;
   AG3.SFC20_1_RET_VAL := 0;
   AG3.SFC20_2_RET_VAL := 0;
   AG3.SFC20_3_RET_VAL := 0;
   AG3.SFC20_4_RET_VAL := 0;
   AG3.SFC20_5_RET_VAL := 0;
   AG3.SFC20_6_RET_VAL := 0;
   AG3.SFC20_7_RET_VAL := 0;
   AG3.SFC20_8_RET_VAL := 0;
   AG3.SFC20_9_RET_VAL := 0;
   AG3.SFC20_10_RET_VAL := 0;
   AG3.SP[0] := W#16#0;
   AG3.SP[1] := W#16#0;
   AG3.SP[2] := W#16#0;
   AG3.SP[3] := W#16#0;
   AG3.SP[4] := W#16#0;
   AG3.SP[5] := W#16#0;
   AG3.SP[6] := W#16#0;
   AG3.SP[7] := W#16#0;
   AG3.SP[8] := W#16#0;
   AG3.SP[9] := W#16#0;
   AG4.FC6_NDR := FALSE;
   AG4.FC6_ERROR := FALSE;
   AG4.SP1 := FALSE;
   AG4.SP2 := FALSE;
   AG4.FC5_NDR := FALSE;
   AG4.FC5_ERROR := FALSE;
   AG4.SP3 := FALSE;
   AG4.SP4 := FALSE;
   AG4.FC6_STATUS := W#16#0;
   AG4.FC6_DPSTATUS := B#16#0;
   AG4.FC5_STATUS := W#16#0;
   AG4.SP5 := W#16#0;
   AG4.SFC20_1_RET_VAL := 0;
   AG4.SFC20_2_RET_VAL := 0;
   AG4.SFC20_3_RET_VAL := 0;
   AG4.SFC20_4_RET_VAL := 0;
   AG4.SFC20_5_RET_VAL := 0;
   AG4.SFC20_6_RET_VAL := 0;
   AG4.SFC20_7_RET_VAL := 0;
   AG4.SFC20_8_RET_VAL := 0;
   AG4.SFC20_9_RET_VAL := 0;
   AG4.SFC20_10_RET_VAL := 0;
   AG4.SP[0] := W#16#0;
   AG4.SP[1] := W#16#0;
   AG4.SP[2] := W#16#0;
   AG4.SP[3] := W#16#0;
   AG4.SP[4] := W#16#0;
   AG4.SP[5] := W#16#0;
   AG4.SP[6] := W#16#0;
   AG4.SP[7] := W#16#0;
   AG4.SP[8] := W#16#0;
   AG4.SP[9] := W#16#0;
   AG5.FC6_NDR := FALSE;
   AG5.FC6_ERROR := FALSE;
   AG5.SP1 := FALSE;
   AG5.SP2 := FALSE;
   AG5.FC5_NDR := FALSE;
   AG5.FC5_ERROR := FALSE;
   AG5.SP3 := FALSE;
   AG5.SP4 := FALSE;
   AG5.FC6_STATUS := W#16#0;
   AG5.FC6_DPSTATUS := B#16#0;
   AG5.FC5_STATUS := W#16#0;
   AG5.SP5 := W#16#0;
   AG5.SFC20_1_RET_VAL := 0;
   AG5.SFC20_2_RET_VAL := 0;
   AG5.SFC20_3_RET_VAL := 0;
   AG5.SFC20_4_RET_VAL := 0;
   AG5.SFC20_5_RET_VAL := 0;
   AG5.SFC20_6_RET_VAL := 0;
   AG5.SFC20_7_RET_VAL := 0;
   AG5.SFC20_8_RET_VAL := 0;
   AG5.SFC20_9_RET_VAL := 0;
   AG5.SFC20_10_RET_VAL := 0;
   AG5.SP[0] := W#16#0;
   AG5.SP[1] := W#16#0;
   AG5.SP[2] := W#16#0;
   AG5.SP[3] := W#16#0;
   AG5.SP[4] := W#16#0;
   AG5.SP[5] := W#16#0;
   AG5.SP[6] := W#16#0;
   AG5.SP[7] := W#16#0;
   AG5.SP[8] := W#16#0;
   AG5.SP[9] := W#16#0;
   AG6.FC6_NDR := FALSE;
   AG6.FC6_ERROR := FALSE;
   AG6.SP1 := FALSE;
   AG6.SP2 := FALSE;
   AG6.FC5_NDR := FALSE;
   AG6.FC5_ERROR := FALSE;
   AG6.SP3 := FALSE;
   AG6.SP4 := FALSE;
   AG6.FC6_STATUS := W#16#0;
   AG6.FC6_DPSTATUS := B#16#0;
   AG6.FC5_STATUS := W#16#0;
   AG6.SP5 := W#16#0;
   AG6.SFC20_1_RET_VAL := 0;
   AG6.SFC20_2_RET_VAL := 0;
   AG6.SFC20_3_RET_VAL := 0;
   AG6.SFC20_4_RET_VAL := 0;
   AG6.SFC20_5_RET_VAL := 0;
   AG6.SFC20_6_RET_VAL := 0;
   AG6.SFC20_7_RET_VAL := 0;
   AG6.SFC20_8_RET_VAL := 0;
   AG6.SFC20_9_RET_VAL := 0;
   AG6.SFC20_10_RET_VAL := 0;
   AG6.SP[0] := W#16#0;
   AG6.SP[1] := W#16#0;
   AG6.SP[2] := W#16#0;
   AG6.SP[3] := W#16#0;
   AG6.SP[4] := W#16#0;
   AG6.SP[5] := W#16#0;
   AG6.SP[6] := W#16#0;
   AG6.SP[7] := W#16#0;
   AG6.SP[8] := W#16#0;
   AG6.SP[9] := W#16#0;
   AG7.FC6_NDR := FALSE;
   AG7.FC6_ERROR := FALSE;
   AG7.SP1 := FALSE;
   AG7.SP2 := FALSE;
   AG7.FC5_NDR := FALSE;
   AG7.FC5_ERROR := FALSE;
   AG7.SP3 := FALSE;
   AG7.SP4 := FALSE;
   AG7.FC6_STATUS := W#16#0;
   AG7.FC6_DPSTATUS := B#16#0;
   AG7.FC5_STATUS := W#16#0;
   AG7.SP5 := W#16#0;
   AG7.SFC20_1_RET_VAL := 0;
   AG7.SFC20_2_RET_VAL := 0;
   AG7.SFC20_3_RET_VAL := 0;
   AG7.SFC20_4_RET_VAL := 0;
   AG7.SFC20_5_RET_VAL := 0;
   AG7.SFC20_6_RET_VAL := 0;
   AG7.SFC20_7_RET_VAL := 0;
   AG7.SFC20_8_RET_VAL := 0;
   AG7.SFC20_9_RET_VAL := 0;
   AG7.SFC20_10_RET_VAL := 0;
   AG7.SP[0] := W#16#0;
   AG7.SP[1] := W#16#0;
   AG7.SP[2] := W#16#0;
   AG7.SP[3] := W#16#0;
   AG7.SP[4] := W#16#0;
   AG7.SP[5] := W#16#0;
   AG7.SP[6] := W#16#0;
   AG7.SP[7] := W#16#0;
   AG7.SP[8] := W#16#0;
   AG7.SP[9] := W#16#0;
   SP[0] := W#16#0;
   SP[1] := W#16#0;
   SP[2] := W#16#0;
   SP[3] := W#16#0;
   SP[4] := W#16#0;
   SP[5] := W#16#0;
   SP[6] := W#16#0;
   SP[7] := W#16#0;
   SP[8] := W#16#0;
   SP[9] := W#16#0;
   SP[10] := W#16#0;
   SP[11] := W#16#0;
   SP[12] := W#16#0;
   SP[13] := W#16#0;
   SP[14] := W#16#0;
   SP[15] := W#16#0;
   SP[16] := W#16#0;
   SP[17] := W#16#0;
   SP[18] := W#16#0;
   SP[19] := W#16#0;
   SP[20] := W#16#0;
   SP[21] := W#16#0;
   SP[22] := W#16#0;
   SP[23] := W#16#0;
   SP[24] := W#16#0;
   SP[25] := W#16#0;
   SP[26] := W#16#0;
   SP[27] := W#16#0;
   SP[28] := W#16#0;
   SP[29] := W#16#0;
   SP[30] := W#16#0;
   SP[31] := W#16#0;
   SP[32] := W#16#0;
   SP[33] := W#16#0;
   SP[34] := W#16#0;
   SP[35] := W#16#0;
   SP[36] := W#16#0;
   SP[37] := W#16#0;
   SP[38] := W#16#0;
   SP[39] := W#16#0;
   SP[40] := W#16#0;
   SP[41] := W#16#0;
   SP[42] := W#16#0;
   SP[43] := W#16#0;
   SP[44] := W#16#0;
   SP[45] := W#16#0;
   SP[46] := W#16#0;
   SP[47] := W#16#0;
   SP[48] := W#16#0;
   SP[49] := W#16#0;
   SP[50] := W#16#0;
   SP[51] := W#16#0;
   SP[52] := W#16#0;
   SP[53] := W#16#0;
   SP[54] := W#16#0;
   SP[55] := W#16#0;
   SP[56] := W#16#0;
   SP[57] := W#16#0;
   SP[58] := W#16#0;
   SP[59] := W#16#0;
   SP[60] := W#16#0;
   SP[61] := W#16#0;
   SP[62] := W#16#0;
   SP[63] := W#16#0;
   SP[64] := W#16#0;
   SP[65] := W#16#0;
   SP[66] := W#16#0;
   SP[67] := W#16#0;
   SP[68] := W#16#0;
   SP[69] := W#16#0;
   SP[70] := W#16#0;
   SP[71] := W#16#0;
   SP[72] := W#16#0;
   SP[73] := W#16#0;
   SP[74] := W#16#0;
   CTYPE_RET_VAL[0] := 0;
   CTYPE_RET_VAL[1] := 0;
   CTYPE_RET_VAL[2] := 0;
   CTYPE_RET_VAL[3] := 0;
   CTYPE_RET_VAL[4] := 0;
   CTYPE_RET_VAL[5] := 0;
   CTYPE_RET_VAL[6] := 0;
   CTYPE_RET_VAL[7] := 0;
   CTYPE_RET_VAL[8] := 0;
   CTYPE_RET_VAL[9] := 0;
   CTYPE_RET_VAL[10] := 0;
   CTYPE_RET_VAL[11] := 0;
   CTYPE_RET_VAL[12] := 0;
   CTYPE_RET_VAL[13] := 0;
   CTYPE_RET_VAL[14] := 0;
   CTYPE_RET_VAL[15] := 0;
   CTYPE_RET_VAL[16] := 0;
   CTYPE_RET_VAL[17] := 0;
   CTYPE_RET_VAL[18] := 0;
   CTYPE_RET_VAL[19] := 0;
   CTYPE_RET_VAL[20] := 0;
   CTYPE_RET_VAL[21] := 0;
   CTYPE_RET_VAL[22] := 0;
   CTYPE_RET_VAL[23] := 0;
   CTYPE_RET_VAL[24] := 0;
   CTYPE_RET_VAL[25] := 0;
   CTYPE_RET_VAL[26] := 0;
   CTYPE_RET_VAL[27] := 0;
   CTYPE_RET_VAL[28] := 0;
   CTYPE_RET_VAL[29] := 0;
   CTYPE_RET_VAL[30] := 0;
   CTYPE_RET_VAL[31] := 0;
   CTYPE_RET_VAL[32] := 0;
   CTYPE_RET_VAL[33] := 0;
   CTYPE_RET_VAL[34] := 0;
   CTYPE_RET_VAL[35] := 0;
   CTYPE_RET_VAL[36] := 0;
   CTYPE_RET_VAL[37] := 0;
   CTYPE_RET_VAL[38] := 0;
   CTYPE_RET_VAL[39] := 0;
   CTYPE_RET_VAL[40] := 0;
   CTYPE_RET_VAL[41] := 0;
   CTYPE_RET_VAL[42] := 0;
   CTYPE_RET_VAL[43] := 0;
   CTYPE_RET_VAL[44] := 0;
   CTYPE_RET_VAL[45] := 0;
   CTYPE_RET_VAL[46] := 0;
   CTYPE_RET_VAL[47] := 0;
   CTYPE_RET_VAL[48] := 0;
   CTYPE_RET_VAL[49] := 0;
   CTYPE_RET_VAL[50] := 0;
   CTYPE_RET_VAL[51] := 0;
   CTYPE_RET_VAL[52] := 0;
   CTYPE_RET_VAL[53] := 0;
   CTYPE_RET_VAL[54] := 0;
   CTYPE_RET_VAL[55] := 0;
   CTYPE_RET_VAL[56] := 0;
   CTYPE_RET_VAL[57] := 0;
   CTYPE_RET_VAL[58] := 0;
   CTYPE_RET_VAL[59] := 0;
   CTYPE_RET_VAL[60] := 0;
   CTYPE_RET_VAL[61] := 0;
   CTYPE_RET_VAL[62] := 0;
   CTYPE_RET_VAL[63] := 0;
   CTYPE_RET_VAL[64] := 0;
   CTYPE_RET_VAL[65] := 0;
   CTYPE_RET_VAL[66] := 0;
   CTYPE_RET_VAL[67] := 0;
   CTYPE_RET_VAL[68] := 0;
   CTYPE_RET_VAL[69] := 0;
   CTYPE_RET_VAL[70] := 0;
   CTYPE_RET_VAL[71] := 0;
   CTYPE_RET_VAL[72] := 0;
   CTYPE_RET_VAL[73] := 0;
   CTYPE_RET_VAL[74] := 0;
   CTYPE_RET_VAL[75] := 0;
   CTYPE_RET_VAL[76] := 0;
   CTYPE_RET_VAL[77] := 0;
   CTYPE_RET_VAL[78] := 0;
   CTYPE_RET_VAL[79] := 0;
   CTYPE_RET_VAL[80] := 0;
   CTYPE_RET_VAL[81] := 0;
   CTYPE_RET_VAL[82] := 0;
   CTYPE_RET_VAL[83] := 0;
   CTYPE_RET_VAL[84] := 0;
   CTYPE_RET_VAL[85] := 0;
   CTYPE_RET_VAL[86] := 0;
   CTYPE_RET_VAL[87] := 0;
   CTYPE_RET_VAL[88] := 0;
   CTYPE_RET_VAL[89] := 0;
   CTYPE_RET_VAL[90] := 0;
   CTYPE_RET_VAL[91] := 0;
   CTYPE_RET_VAL[92] := 0;
   CTYPE_RET_VAL[93] := 0;
   CTYPE_RET_VAL[94] := 0;
   CTYPE_RET_VAL[95] := 0;
   CTYPE_RET_VAL[96] := 0;
   CTYPE_RET_VAL[97] := 0;
   CTYPE_RET_VAL[98] := 0;
   CTYPE_RET_VAL[99] := 0;
   MES_RET_VAL1[0] := 0;
   MES_RET_VAL1[1] := 0;
   MES_RET_VAL1[2] := 0;
   MES_RET_VAL1[3] := 0;
   MES_RET_VAL1[4] := 0;
   MES_RET_VAL1[5] := 0;
   MES_RET_VAL1[6] := 0;
   MES_RET_VAL1[7] := 0;
   MES_RET_VAL1[8] := 0;
   MES_RET_VAL1[9] := 0;
   MES_RET_VAL1[10] := 0;
   MES_RET_VAL1[11] := 0;
   MES_RET_VAL1[12] := 0;
   MES_RET_VAL1[13] := 0;
   MES_RET_VAL1[14] := 0;
   MES_RET_VAL1[15] := 0;
   MES_RET_VAL1[16] := 0;
   MES_RET_VAL1[17] := 0;
   MES_RET_VAL1[18] := 0;
   MES_RET_VAL1[19] := 0;
   MES_RET_VAL1[20] := 0;
   MES_RET_VAL1[21] := 0;
   MES_RET_VAL1[22] := 0;
   MES_RET_VAL1[23] := 0;
   MES_RET_VAL1[24] := 0;
   MES_RET_VAL1[25] := 0;
   MES_RET_VAL1[26] := 0;
   MES_RET_VAL1[27] := 0;
   MES_RET_VAL1[28] := 0;
   MES_RET_VAL1[29] := 0;
   MES_RET_VAL1[30] := 0;
   MES_RET_VAL1[31] := 0;
   MES_RET_VAL1[32] := 0;
   MES_RET_VAL1[33] := 0;
   MES_RET_VAL1[34] := 0;
   MES_RET_VAL1[35] := 0;
   MES_RET_VAL1[36] := 0;
   MES_RET_VAL1[37] := 0;
   MES_RET_VAL1[38] := 0;
   MES_RET_VAL1[39] := 0;
   MES_RET_VAL1[40] := 0;
   MES_RET_VAL1[41] := 0;
   MES_RET_VAL1[42] := 0;
   MES_RET_VAL1[43] := 0;
   MES_RET_VAL1[44] := 0;
   MES_RET_VAL1[45] := 0;
   MES_RET_VAL1[46] := 0;
   MES_RET_VAL1[47] := 0;
   MES_RET_VAL1[48] := 0;
   MES_RET_VAL1[49] := 0;
   MES_RET_VAL1[50] := 0;
   MES_RET_VAL1[51] := 0;
   MES_RET_VAL1[52] := 0;
   MES_RET_VAL1[53] := 0;
   MES_RET_VAL1[54] := 0;
   MES_RET_VAL1[55] := 0;
   MES_RET_VAL1[56] := 0;
   MES_RET_VAL1[57] := 0;
   MES_RET_VAL1[58] := 0;
   MES_RET_VAL1[59] := 0;
   MES_RET_VAL1[60] := 0;
   MES_RET_VAL1[61] := 0;
   MES_RET_VAL1[62] := 0;
   MES_RET_VAL1[63] := 0;
   MES_RET_VAL1[64] := 0;
   MES_RET_VAL1[65] := 0;
   MES_RET_VAL1[66] := 0;
   MES_RET_VAL1[67] := 0;
   MES_RET_VAL1[68] := 0;
   MES_RET_VAL1[69] := 0;
   MES_RET_VAL1[70] := 0;
   MES_RET_VAL1[71] := 0;
   MES_RET_VAL1[72] := 0;
   MES_RET_VAL1[73] := 0;
   MES_RET_VAL1[74] := 0;
   MES_RET_VAL1[75] := 0;
   MES_RET_VAL1[76] := 0;
   MES_RET_VAL1[77] := 0;
   MES_RET_VAL1[78] := 0;
   MES_RET_VAL1[79] := 0;
   MES_RET_VAL1[80] := 0;
   MES_RET_VAL1[81] := 0;
   MES_RET_VAL1[82] := 0;
   MES_RET_VAL1[83] := 0;
   MES_RET_VAL1[84] := 0;
   MES_RET_VAL1[85] := 0;
   MES_RET_VAL1[86] := 0;
   MES_RET_VAL1[87] := 0;
   MES_RET_VAL1[88] := 0;
   MES_RET_VAL1[89] := 0;
   MES_RET_VAL1[90] := 0;
   MES_RET_VAL1[91] := 0;
   MES_RET_VAL1[92] := 0;
   MES_RET_VAL1[93] := 0;
   MES_RET_VAL1[94] := 0;
   MES_RET_VAL1[95] := 0;
   MES_RET_VAL1[96] := 0;
   MES_RET_VAL1[97] := 0;
   MES_RET_VAL1[98] := 0;
   MES_RET_VAL1[99] := 0;
   MES_RET_VAL1[100] := 0;
   MES_RET_VAL1[101] := 0;
   MES_RET_VAL1[102] := 0;
   MES_RET_VAL1[103] := 0;
   MES_RET_VAL1[104] := 0;
   MES_RET_VAL1[105] := 0;
   MES_RET_VAL1[106] := 0;
   MES_RET_VAL1[107] := 0;
   MES_RET_VAL1[108] := 0;
   MES_RET_VAL1[109] := 0;
   MES_RET_VAL1[110] := 0;
   MES_RET_VAL1[111] := 0;
   MES_RET_VAL1[112] := 0;
   MES_RET_VAL1[113] := 0;
   MES_RET_VAL1[114] := 0;
   MES_RET_VAL1[115] := 0;
   MES_RET_VAL1[116] := 0;
   MES_RET_VAL1[117] := 0;
   MES_RET_VAL1[118] := 0;
   MES_RET_VAL1[119] := 0;
   MES_RET_VAL1[120] := 0;
   MES_RET_VAL1[121] := 0;
   MES_RET_VAL1[122] := 0;
   MES_RET_VAL1[123] := 0;
   MES_RET_VAL1[124] := 0;
   MES_RET_VAL1[125] := 0;
   MES_RET_VAL1[126] := 0;
   MES_RET_VAL1[127] := 0;
   MES_RET_VAL1[128] := 0;
   MES_RET_VAL1[129] := 0;
   MES_RET_VAL1[130] := 0;
   MES_RET_VAL1[131] := 0;
   MES_RET_VAL1[132] := 0;
   MES_RET_VAL1[133] := 0;
   MES_RET_VAL1[134] := 0;
   MES_RET_VAL1[135] := 0;
   MES_RET_VAL1[136] := 0;
   MES_RET_VAL1[137] := 0;
   MES_RET_VAL1[138] := 0;
   MES_RET_VAL1[139] := 0;
   MES_RET_VAL1[140] := 0;
   MES_RET_VAL1[141] := 0;
   MES_RET_VAL1[142] := 0;
   MES_RET_VAL1[143] := 0;
   MES_RET_VAL1[144] := 0;
   MES_RET_VAL1[145] := 0;
   MES_RET_VAL1[146] := 0;
   MES_RET_VAL1[147] := 0;
   MES_RET_VAL1[148] := 0;
   MES_RET_VAL1[149] := 0;
   MES_RET_VAL1[150] := 0;
   MES_RET_VAL1[151] := 0;
   MES_RET_VAL1[152] := 0;
   MES_RET_VAL1[153] := 0;
   MES_RET_VAL1[154] := 0;
   MES_RET_VAL1[155] := 0;
   MES_RET_VAL1[156] := 0;
   MES_RET_VAL1[157] := 0;
   MES_RET_VAL1[158] := 0;
   MES_RET_VAL1[159] := 0;
   MES_RET_VAL1[160] := 0;
   MES_RET_VAL1[161] := 0;
   MES_RET_VAL1[162] := 0;
   MES_RET_VAL1[163] := 0;
   MES_RET_VAL1[164] := 0;
   MES_RET_VAL1[165] := 0;
   MES_RET_VAL1[166] := 0;
   MES_RET_VAL1[167] := 0;
   MES_RET_VAL1[168] := 0;
   MES_RET_VAL1[169] := 0;
   MES_RET_VAL1[170] := 0;
   MES_RET_VAL1[171] := 0;
   MES_RET_VAL1[172] := 0;
   MES_RET_VAL1[173] := 0;
   MES_RET_VAL1[174] := 0;
   MES_RET_VAL1[175] := 0;
   MES_RET_VAL1[176] := 0;
   MES_RET_VAL1[177] := 0;
   MES_RET_VAL1[178] := 0;
   MES_RET_VAL1[179] := 0;
   MES_RET_VAL1[180] := 0;
   MES_RET_VAL1[181] := 0;
   MES_RET_VAL1[182] := 0;
   MES_RET_VAL1[183] := 0;
   MES_RET_VAL1[184] := 0;
   MES_RET_VAL1[185] := 0;
   MES_RET_VAL1[186] := 0;
   MES_RET_VAL1[187] := 0;
   MES_RET_VAL1[188] := 0;
   MES_RET_VAL1[189] := 0;
   MES_RET_VAL1[190] := 0;
   MES_RET_VAL1[191] := 0;
   MES_RET_VAL1[192] := 0;
   MES_RET_VAL1[193] := 0;
   MES_RET_VAL1[194] := 0;
   MES_RET_VAL1[195] := 0;
   MES_RET_VAL1[196] := 0;
   MES_RET_VAL1[197] := 0;
   MES_RET_VAL1[198] := 0;
   MES_RET_VAL1[199] := 0;
END_DATA_BLOCK

DATA_BLOCK DB 60
TITLE =
VERSION : 0.1


  STRUCT
   FC1_SEND_1 : ARRAY  [0 .. 499 ] OF BYTE  := B#16#0;
  END_STRUCT ;
BEGIN
   FC1_SEND_1[0] := B#16#0;
   FC1_SEND_1[1] := B#16#0;
   FC1_SEND_1[2] := B#16#0;
   FC1_SEND_1[3] := B#16#0;
   FC1_SEND_1[4] := B#16#0;
   FC1_SEND_1[5] := B#16#0;
   FC1_SEND_1[6] := B#16#0;
   FC1_SEND_1[7] := B#16#0;
   FC1_SEND_1[8] := B#16#0;
   FC1_SEND_1[9] := B#16#0;
   FC1_SEND_1[10] := B#16#0;
   FC1_SEND_1[11] := B#16#0;
   FC1_SEND_1[12] := B#16#0;
   FC1_SEND_1[13] := B#16#0;
   FC1_SEND_1[14] := B#16#0;
   FC1_SEND_1[15] := B#16#0;
   FC1_SEND_1[16] := B#16#0;
   FC1_SEND_1[17] := B#16#0;
   FC1_SEND_1[18] := B#16#0;
   FC1_SEND_1[19] := B#16#0;
   FC1_SEND_1[20] := B#16#0;
   FC1_SEND_1[21] := B#16#0;
   FC1_SEND_1[22] := B#16#0;
   FC1_SEND_1[23] := B#16#0;
   FC1_SEND_1[24] := B#16#0;
   FC1_SEND_1[25] := B#16#0;
   FC1_SEND_1[26] := B#16#0;
   FC1_SEND_1[27] := B#16#0;
   FC1_SEND_1[28] := B#16#0;
   FC1_SEND_1[29] := B#16#0;
   FC1_SEND_1[30] := B#16#0;
   FC1_SEND_1[31] := B#16#0;
   FC1_SEND_1[32] := B#16#0;
   FC1_SEND_1[33] := B#16#0;
   FC1_SEND_1[34] := B#16#0;
   FC1_SEND_1[35] := B#16#0;
   FC1_SEND_1[36] := B#16#0;
   FC1_SEND_1[37] := B#16#0;
   FC1_SEND_1[38] := B#16#0;
   FC1_SEND_1[39] := B#16#0;
   FC1_SEND_1[40] := B#16#0;
   FC1_SEND_1[41] := B#16#0;
   FC1_SEND_1[42] := B#16#0;
   FC1_SEND_1[43] := B#16#0;
   FC1_SEND_1[44] := B#16#0;
   FC1_SEND_1[45] := B#16#0;
   FC1_SEND_1[46] := B#16#0;
   FC1_SEND_1[47] := B#16#0;
   FC1_SEND_1[48] := B#16#0;
   FC1_SEND_1[49] := B#16#0;
   FC1_SEND_1[50] := B#16#0;
   FC1_SEND_1[51] := B#16#0;
   FC1_SEND_1[52] := B#16#0;
   FC1_SEND_1[53] := B#16#0;
   FC1_SEND_1[54] := B#16#0;
   FC1_SEND_1[55] := B#16#0;
   FC1_SEND_1[56] := B#16#0;
   FC1_SEND_1[57] := B#16#0;
   FC1_SEND_1[58] := B#16#0;
   FC1_SEND_1[59] := B#16#0;
   FC1_SEND_1[60] := B#16#0;
   FC1_SEND_1[61] := B#16#0;
   FC1_SEND_1[62] := B#16#0;
   FC1_SEND_1[63] := B#16#0;
   FC1_SEND_1[64] := B#16#0;
   FC1_SEND_1[65] := B#16#0;
   FC1_SEND_1[66] := B#16#0;
   FC1_SEND_1[67] := B#16#0;
   FC1_SEND_1[68] := B#16#0;
   FC1_SEND_1[69] := B#16#0;
   FC1_SEND_1[70] := B#16#0;
   FC1_SEND_1[71] := B#16#0;
   FC1_SEND_1[72] := B#16#0;
   FC1_SEND_1[73] := B#16#0;
   FC1_SEND_1[74] := B#16#0;
   FC1_SEND_1[75] := B#16#0;
   FC1_SEND_1[76] := B#16#0;
   FC1_SEND_1[77] := B#16#0;
   FC1_SEND_1[78] := B#16#0;
   FC1_SEND_1[79] := B#16#0;
   FC1_SEND_1[80] := B#16#0;
   FC1_SEND_1[81] := B#16#0;
   FC1_SEND_1[82] := B#16#0;
   FC1_SEND_1[83] := B#16#0;
   FC1_SEND_1[84] := B#16#0;
   FC1_SEND_1[85] := B#16#0;
   FC1_SEND_1[86] := B#16#0;
   FC1_SEND_1[87] := B#16#0;
   FC1_SEND_1[88] := B#16#0;
   FC1_SEND_1[89] := B#16#0;
   FC1_SEND_1[90] := B#16#0;
   FC1_SEND_1[91] := B#16#0;
   FC1_SEND_1[92] := B#16#0;
   FC1_SEND_1[93] := B#16#0;
   FC1_SEND_1[94] := B#16#0;
   FC1_SEND_1[95] := B#16#0;
   FC1_SEND_1[96] := B#16#0;
   FC1_SEND_1[97] := B#16#0;
   FC1_SEND_1[98] := B#16#0;
   FC1_SEND_1[99] := B#16#0;
   FC1_SEND_1[100] := B#16#0;
   FC1_SEND_1[101] := B#16#0;
   FC1_SEND_1[102] := B#16#0;
   FC1_SEND_1[103] := B#16#0;
   FC1_SEND_1[104] := B#16#0;
   FC1_SEND_1[105] := B#16#0;
   FC1_SEND_1[106] := B#16#0;
   FC1_SEND_1[107] := B#16#0;
   FC1_SEND_1[108] := B#16#0;
   FC1_SEND_1[109] := B#16#0;
   FC1_SEND_1[110] := B#16#0;
   FC1_SEND_1[111] := B#16#0;
   FC1_SEND_1[112] := B#16#0;
   FC1_SEND_1[113] := B#16#0;
   FC1_SEND_1[114] := B#16#0;
   FC1_SEND_1[115] := B#16#0;
   FC1_SEND_1[116] := B#16#0;
   FC1_SEND_1[117] := B#16#0;
   FC1_SEND_1[118] := B#16#0;
   FC1_SEND_1[119] := B#16#0;
   FC1_SEND_1[120] := B#16#0;
   FC1_SEND_1[121] := B#16#0;
   FC1_SEND_1[122] := B#16#0;
   FC1_SEND_1[123] := B#16#0;
   FC1_SEND_1[124] := B#16#0;
   FC1_SEND_1[125] := B#16#0;
   FC1_SEND_1[126] := B#16#0;
   FC1_SEND_1[127] := B#16#0;
   FC1_SEND_1[128] := B#16#0;
   FC1_SEND_1[129] := B#16#0;
   FC1_SEND_1[130] := B#16#0;
   FC1_SEND_1[131] := B#16#0;
   FC1_SEND_1[132] := B#16#0;
   FC1_SEND_1[133] := B#16#0;
   FC1_SEND_1[134] := B#16#0;
   FC1_SEND_1[135] := B#16#0;
   FC1_SEND_1[136] := B#16#0;
   FC1_SEND_1[137] := B#16#0;
   FC1_SEND_1[138] := B#16#0;
   FC1_SEND_1[139] := B#16#0;
   FC1_SEND_1[140] := B#16#0;
   FC1_SEND_1[141] := B#16#0;
   FC1_SEND_1[142] := B#16#0;
   FC1_SEND_1[143] := B#16#0;
   FC1_SEND_1[144] := B#16#0;
   FC1_SEND_1[145] := B#16#0;
   FC1_SEND_1[146] := B#16#0;
   FC1_SEND_1[147] := B#16#0;
   FC1_SEND_1[148] := B#16#0;
   FC1_SEND_1[149] := B#16#0;
   FC1_SEND_1[150] := B#16#0;
   FC1_SEND_1[151] := B#16#0;
   FC1_SEND_1[152] := B#16#0;
   FC1_SEND_1[153] := B#16#0;
   FC1_SEND_1[154] := B#16#0;
   FC1_SEND_1[155] := B#16#0;
   FC1_SEND_1[156] := B#16#0;
   FC1_SEND_1[157] := B#16#0;
   FC1_SEND_1[158] := B#16#0;
   FC1_SEND_1[159] := B#16#0;
   FC1_SEND_1[160] := B#16#0;
   FC1_SEND_1[161] := B#16#0;
   FC1_SEND_1[162] := B#16#0;
   FC1_SEND_1[163] := B#16#0;
   FC1_SEND_1[164] := B#16#0;
   FC1_SEND_1[165] := B#16#0;
   FC1_SEND_1[166] := B#16#0;
   FC1_SEND_1[167] := B#16#0;
   FC1_SEND_1[168] := B#16#0;
   FC1_SEND_1[169] := B#16#0;
   FC1_SEND_1[170] := B#16#0;
   FC1_SEND_1[171] := B#16#0;
   FC1_SEND_1[172] := B#16#0;
   FC1_SEND_1[173] := B#16#0;
   FC1_SEND_1[174] := B#16#0;
   FC1_SEND_1[175] := B#16#0;
   FC1_SEND_1[176] := B#16#0;
   FC1_SEND_1[177] := B#16#0;
   FC1_SEND_1[178] := B#16#0;
   FC1_SEND_1[179] := B#16#0;
   FC1_SEND_1[180] := B#16#0;
   FC1_SEND_1[181] := B#16#0;
   FC1_SEND_1[182] := B#16#0;
   FC1_SEND_1[183] := B#16#0;
   FC1_SEND_1[184] := B#16#0;
   FC1_SEND_1[185] := B#16#0;
   FC1_SEND_1[186] := B#16#0;
   FC1_SEND_1[187] := B#16#0;
   FC1_SEND_1[188] := B#16#0;
   FC1_SEND_1[189] := B#16#0;
   FC1_SEND_1[190] := B#16#0;
   FC1_SEND_1[191] := B#16#0;
   FC1_SEND_1[192] := B#16#0;
   FC1_SEND_1[193] := B#16#0;
   FC1_SEND_1[194] := B#16#0;
   FC1_SEND_1[195] := B#16#0;
   FC1_SEND_1[196] := B#16#0;
   FC1_SEND_1[197] := B#16#0;
   FC1_SEND_1[198] := B#16#0;
   FC1_SEND_1[199] := B#16#0;
   FC1_SEND_1[200] := B#16#0;
   FC1_SEND_1[201] := B#16#0;
   FC1_SEND_1[202] := B#16#0;
   FC1_SEND_1[203] := B#16#0;
   FC1_SEND_1[204] := B#16#0;
   FC1_SEND_1[205] := B#16#0;
   FC1_SEND_1[206] := B#16#0;
   FC1_SEND_1[207] := B#16#0;
   FC1_SEND_1[208] := B#16#0;
   FC1_SEND_1[209] := B#16#0;
   FC1_SEND_1[210] := B#16#0;
   FC1_SEND_1[211] := B#16#0;
   FC1_SEND_1[212] := B#16#0;
   FC1_SEND_1[213] := B#16#0;
   FC1_SEND_1[214] := B#16#0;
   FC1_SEND_1[215] := B#16#0;
   FC1_SEND_1[216] := B#16#0;
   FC1_SEND_1[217] := B#16#0;
   FC1_SEND_1[218] := B#16#0;
   FC1_SEND_1[219] := B#16#0;
   FC1_SEND_1[220] := B#16#0;
   FC1_SEND_1[221] := B#16#0;
   FC1_SEND_1[222] := B#16#0;
   FC1_SEND_1[223] := B#16#0;
   FC1_SEND_1[224] := B#16#0;
   FC1_SEND_1[225] := B#16#0;
   FC1_SEND_1[226] := B#16#0;
   FC1_SEND_1[227] := B#16#0;
   FC1_SEND_1[228] := B#16#0;
   FC1_SEND_1[229] := B#16#0;
   FC1_SEND_1[230] := B#16#0;
   FC1_SEND_1[231] := B#16#0;
   FC1_SEND_1[232] := B#16#0;
   FC1_SEND_1[233] := B#16#0;
   FC1_SEND_1[234] := B#16#0;
   FC1_SEND_1[235] := B#16#0;
   FC1_SEND_1[236] := B#16#0;
   FC1_SEND_1[237] := B#16#0;
   FC1_SEND_1[238] := B#16#0;
   FC1_SEND_1[239] := B#16#0;
   FC1_SEND_1[240] := B#16#0;
   FC1_SEND_1[241] := B#16#0;
   FC1_SEND_1[242] := B#16#0;
   FC1_SEND_1[243] := B#16#0;
   FC1_SEND_1[244] := B#16#0;
   FC1_SEND_1[245] := B#16#0;
   FC1_SEND_1[246] := B#16#0;
   FC1_SEND_1[247] := B#16#0;
   FC1_SEND_1[248] := B#16#0;
   FC1_SEND_1[249] := B#16#0;
   FC1_SEND_1[250] := B#16#0;
   FC1_SEND_1[251] := B#16#0;
   FC1_SEND_1[252] := B#16#0;
   FC1_SEND_1[253] := B#16#0;
   FC1_SEND_1[254] := B#16#0;
   FC1_SEND_1[255] := B#16#0;
   FC1_SEND_1[256] := B#16#0;
   FC1_SEND_1[257] := B#16#0;
   FC1_SEND_1[258] := B#16#0;
   FC1_SEND_1[259] := B#16#0;
   FC1_SEND_1[260] := B#16#0;
   FC1_SEND_1[261] := B#16#0;
   FC1_SEND_1[262] := B#16#0;
   FC1_SEND_1[263] := B#16#0;
   FC1_SEND_1[264] := B#16#0;
   FC1_SEND_1[265] := B#16#0;
   FC1_SEND_1[266] := B#16#0;
   FC1_SEND_1[267] := B#16#0;
   FC1_SEND_1[268] := B#16#0;
   FC1_SEND_1[269] := B#16#0;
   FC1_SEND_1[270] := B#16#0;
   FC1_SEND_1[271] := B#16#0;
   FC1_SEND_1[272] := B#16#0;
   FC1_SEND_1[273] := B#16#0;
   FC1_SEND_1[274] := B#16#0;
   FC1_SEND_1[275] := B#16#0;
   FC1_SEND_1[276] := B#16#0;
   FC1_SEND_1[277] := B#16#0;
   FC1_SEND_1[278] := B#16#0;
   FC1_SEND_1[279] := B#16#0;
   FC1_SEND_1[280] := B#16#0;
   FC1_SEND_1[281] := B#16#0;
   FC1_SEND_1[282] := B#16#0;
   FC1_SEND_1[283] := B#16#0;
   FC1_SEND_1[284] := B#16#0;
   FC1_SEND_1[285] := B#16#0;
   FC1_SEND_1[286] := B#16#0;
   FC1_SEND_1[287] := B#16#0;
   FC1_SEND_1[288] := B#16#0;
   FC1_SEND_1[289] := B#16#0;
   FC1_SEND_1[290] := B#16#0;
   FC1_SEND_1[291] := B#16#0;
   FC1_SEND_1[292] := B#16#0;
   FC1_SEND_1[293] := B#16#0;
   FC1_SEND_1[294] := B#16#0;
   FC1_SEND_1[295] := B#16#0;
   FC1_SEND_1[296] := B#16#0;
   FC1_SEND_1[297] := B#16#0;
   FC1_SEND_1[298] := B#16#0;
   FC1_SEND_1[299] := B#16#0;
   FC1_SEND_1[300] := B#16#0;
   FC1_SEND_1[301] := B#16#0;
   FC1_SEND_1[302] := B#16#0;
   FC1_SEND_1[303] := B#16#0;
   FC1_SEND_1[304] := B#16#0;
   FC1_SEND_1[305] := B#16#0;
   FC1_SEND_1[306] := B#16#0;
   FC1_SEND_1[307] := B#16#0;
   FC1_SEND_1[308] := B#16#0;
   FC1_SEND_1[309] := B#16#0;
   FC1_SEND_1[310] := B#16#0;
   FC1_SEND_1[311] := B#16#0;
   FC1_SEND_1[312] := B#16#0;
   FC1_SEND_1[313] := B#16#0;
   FC1_SEND_1[314] := B#16#0;
   FC1_SEND_1[315] := B#16#0;
   FC1_SEND_1[316] := B#16#0;
   FC1_SEND_1[317] := B#16#0;
   FC1_SEND_1[318] := B#16#0;
   FC1_SEND_1[319] := B#16#0;
   FC1_SEND_1[320] := B#16#0;
   FC1_SEND_1[321] := B#16#0;
   FC1_SEND_1[322] := B#16#0;
   FC1_SEND_1[323] := B#16#0;
   FC1_SEND_1[324] := B#16#0;
   FC1_SEND_1[325] := B#16#0;
   FC1_SEND_1[326] := B#16#0;
   FC1_SEND_1[327] := B#16#0;
   FC1_SEND_1[328] := B#16#0;
   FC1_SEND_1[329] := B#16#0;
   FC1_SEND_1[330] := B#16#0;
   FC1_SEND_1[331] := B#16#0;
   FC1_SEND_1[332] := B#16#0;
   FC1_SEND_1[333] := B#16#0;
   FC1_SEND_1[334] := B#16#0;
   FC1_SEND_1[335] := B#16#0;
   FC1_SEND_1[336] := B#16#0;
   FC1_SEND_1[337] := B#16#0;
   FC1_SEND_1[338] := B#16#0;
   FC1_SEND_1[339] := B#16#0;
   FC1_SEND_1[340] := B#16#0;
   FC1_SEND_1[341] := B#16#0;
   FC1_SEND_1[342] := B#16#0;
   FC1_SEND_1[343] := B#16#0;
   FC1_SEND_1[344] := B#16#0;
   FC1_SEND_1[345] := B#16#0;
   FC1_SEND_1[346] := B#16#0;
   FC1_SEND_1[347] := B#16#0;
   FC1_SEND_1[348] := B#16#0;
   FC1_SEND_1[349] := B#16#0;
   FC1_SEND_1[350] := B#16#0;
   FC1_SEND_1[351] := B#16#0;
   FC1_SEND_1[352] := B#16#0;
   FC1_SEND_1[353] := B#16#0;
   FC1_SEND_1[354] := B#16#0;
   FC1_SEND_1[355] := B#16#0;
   FC1_SEND_1[356] := B#16#0;
   FC1_SEND_1[357] := B#16#0;
   FC1_SEND_1[358] := B#16#0;
   FC1_SEND_1[359] := B#16#0;
   FC1_SEND_1[360] := B#16#0;
   FC1_SEND_1[361] := B#16#0;
   FC1_SEND_1[362] := B#16#0;
   FC1_SEND_1[363] := B#16#0;
   FC1_SEND_1[364] := B#16#0;
   FC1_SEND_1[365] := B#16#0;
   FC1_SEND_1[366] := B#16#0;
   FC1_SEND_1[367] := B#16#0;
   FC1_SEND_1[368] := B#16#0;
   FC1_SEND_1[369] := B#16#0;
   FC1_SEND_1[370] := B#16#0;
   FC1_SEND_1[371] := B#16#0;
   FC1_SEND_1[372] := B#16#0;
   FC1_SEND_1[373] := B#16#0;
   FC1_SEND_1[374] := B#16#0;
   FC1_SEND_1[375] := B#16#0;
   FC1_SEND_1[376] := B#16#0;
   FC1_SEND_1[377] := B#16#0;
   FC1_SEND_1[378] := B#16#0;
   FC1_SEND_1[379] := B#16#0;
   FC1_SEND_1[380] := B#16#0;
   FC1_SEND_1[381] := B#16#0;
   FC1_SEND_1[382] := B#16#0;
   FC1_SEND_1[383] := B#16#0;
   FC1_SEND_1[384] := B#16#0;
   FC1_SEND_1[385] := B#16#0;
   FC1_SEND_1[386] := B#16#0;
   FC1_SEND_1[387] := B#16#0;
   FC1_SEND_1[388] := B#16#0;
   FC1_SEND_1[389] := B#16#0;
   FC1_SEND_1[390] := B#16#0;
   FC1_SEND_1[391] := B#16#0;
   FC1_SEND_1[392] := B#16#0;
   FC1_SEND_1[393] := B#16#0;
   FC1_SEND_1[394] := B#16#0;
   FC1_SEND_1[395] := B#16#0;
   FC1_SEND_1[396] := B#16#0;
   FC1_SEND_1[397] := B#16#0;
   FC1_SEND_1[398] := B#16#0;
   FC1_SEND_1[399] := B#16#0;
   FC1_SEND_1[400] := B#16#0;
   FC1_SEND_1[401] := B#16#0;
   FC1_SEND_1[402] := B#16#0;
   FC1_SEND_1[403] := B#16#0;
   FC1_SEND_1[404] := B#16#0;
   FC1_SEND_1[405] := B#16#0;
   FC1_SEND_1[406] := B#16#0;
   FC1_SEND_1[407] := B#16#0;
   FC1_SEND_1[408] := B#16#0;
   FC1_SEND_1[409] := B#16#0;
   FC1_SEND_1[410] := B#16#0;
   FC1_SEND_1[411] := B#16#0;
   FC1_SEND_1[412] := B#16#0;
   FC1_SEND_1[413] := B#16#0;
   FC1_SEND_1[414] := B#16#0;
   FC1_SEND_1[415] := B#16#0;
   FC1_SEND_1[416] := B#16#0;
   FC1_SEND_1[417] := B#16#0;
   FC1_SEND_1[418] := B#16#0;
   FC1_SEND_1[419] := B#16#0;
   FC1_SEND_1[420] := B#16#0;
   FC1_SEND_1[421] := B#16#0;
   FC1_SEND_1[422] := B#16#0;
   FC1_SEND_1[423] := B#16#0;
   FC1_SEND_1[424] := B#16#0;
   FC1_SEND_1[425] := B#16#0;
   FC1_SEND_1[426] := B#16#0;
   FC1_SEND_1[427] := B#16#0;
   FC1_SEND_1[428] := B#16#0;
   FC1_SEND_1[429] := B#16#0;
   FC1_SEND_1[430] := B#16#0;
   FC1_SEND_1[431] := B#16#0;
   FC1_SEND_1[432] := B#16#0;
   FC1_SEND_1[433] := B#16#0;
   FC1_SEND_1[434] := B#16#0;
   FC1_SEND_1[435] := B#16#0;
   FC1_SEND_1[436] := B#16#0;
   FC1_SEND_1[437] := B#16#0;
   FC1_SEND_1[438] := B#16#0;
   FC1_SEND_1[439] := B#16#0;
   FC1_SEND_1[440] := B#16#0;
   FC1_SEND_1[441] := B#16#0;
   FC1_SEND_1[442] := B#16#0;
   FC1_SEND_1[443] := B#16#0;
   FC1_SEND_1[444] := B#16#0;
   FC1_SEND_1[445] := B#16#0;
   FC1_SEND_1[446] := B#16#0;
   FC1_SEND_1[447] := B#16#0;
   FC1_SEND_1[448] := B#16#0;
   FC1_SEND_1[449] := B#16#0;
   FC1_SEND_1[450] := B#16#0;
   FC1_SEND_1[451] := B#16#0;
   FC1_SEND_1[452] := B#16#0;
   FC1_SEND_1[453] := B#16#0;
   FC1_SEND_1[454] := B#16#0;
   FC1_SEND_1[455] := B#16#0;
   FC1_SEND_1[456] := B#16#0;
   FC1_SEND_1[457] := B#16#0;
   FC1_SEND_1[458] := B#16#0;
   FC1_SEND_1[459] := B#16#0;
   FC1_SEND_1[460] := B#16#0;
   FC1_SEND_1[461] := B#16#0;
   FC1_SEND_1[462] := B#16#0;
   FC1_SEND_1[463] := B#16#0;
   FC1_SEND_1[464] := B#16#0;
   FC1_SEND_1[465] := B#16#0;
   FC1_SEND_1[466] := B#16#0;
   FC1_SEND_1[467] := B#16#0;
   FC1_SEND_1[468] := B#16#0;
   FC1_SEND_1[469] := B#16#0;
   FC1_SEND_1[470] := B#16#0;
   FC1_SEND_1[471] := B#16#0;
   FC1_SEND_1[472] := B#16#0;
   FC1_SEND_1[473] := B#16#0;
   FC1_SEND_1[474] := B#16#0;
   FC1_SEND_1[475] := B#16#0;
   FC1_SEND_1[476] := B#16#0;
   FC1_SEND_1[477] := B#16#0;
   FC1_SEND_1[478] := B#16#0;
   FC1_SEND_1[479] := B#16#0;
   FC1_SEND_1[480] := B#16#0;
   FC1_SEND_1[481] := B#16#0;
   FC1_SEND_1[482] := B#16#0;
   FC1_SEND_1[483] := B#16#0;
   FC1_SEND_1[484] := B#16#0;
   FC1_SEND_1[485] := B#16#0;
   FC1_SEND_1[486] := B#16#0;
   FC1_SEND_1[487] := B#16#0;
   FC1_SEND_1[488] := B#16#0;
   FC1_SEND_1[489] := B#16#0;
   FC1_SEND_1[490] := B#16#0;
   FC1_SEND_1[491] := B#16#0;
   FC1_SEND_1[492] := B#16#0;
   FC1_SEND_1[493] := B#16#0;
   FC1_SEND_1[494] := B#16#0;
   FC1_SEND_1[495] := B#16#0;
   FC1_SEND_1[496] := B#16#0;
   FC1_SEND_1[497] := B#16#0;
   FC1_SEND_1[498] := B#16#0;
   FC1_SEND_1[499] := B#16#0;
END_DATA_BLOCK

DATA_BLOCK DB 61
TITLE =
VERSION : 0.1


  STRUCT
   FC2_RECV_1 : ARRAY  [0 .. 499 ] OF BYTE  := B#16#0;
  END_STRUCT ;
BEGIN
   FC2_RECV_1[0] := B#16#0;
   FC2_RECV_1[1] := B#16#0;
   FC2_RECV_1[2] := B#16#0;
   FC2_RECV_1[3] := B#16#0;
   FC2_RECV_1[4] := B#16#0;
   FC2_RECV_1[5] := B#16#0;
   FC2_RECV_1[6] := B#16#0;
   FC2_RECV_1[7] := B#16#0;
   FC2_RECV_1[8] := B#16#0;
   FC2_RECV_1[9] := B#16#0;
   FC2_RECV_1[10] := B#16#0;
   FC2_RECV_1[11] := B#16#0;
   FC2_RECV_1[12] := B#16#0;
   FC2_RECV_1[13] := B#16#0;
   FC2_RECV_1[14] := B#16#0;
   FC2_RECV_1[15] := B#16#0;
   FC2_RECV_1[16] := B#16#0;
   FC2_RECV_1[17] := B#16#0;
   FC2_RECV_1[18] := B#16#0;
   FC2_RECV_1[19] := B#16#0;
   FC2_RECV_1[20] := B#16#0;
   FC2_RECV_1[21] := B#16#0;
   FC2_RECV_1[22] := B#16#0;
   FC2_RECV_1[23] := B#16#0;
   FC2_RECV_1[24] := B#16#0;
   FC2_RECV_1[25] := B#16#0;
   FC2_RECV_1[26] := B#16#0;
   FC2_RECV_1[27] := B#16#0;
   FC2_RECV_1[28] := B#16#0;
   FC2_RECV_1[29] := B#16#0;
   FC2_RECV_1[30] := B#16#0;
   FC2_RECV_1[31] := B#16#0;
   FC2_RECV_1[32] := B#16#0;
   FC2_RECV_1[33] := B#16#0;
   FC2_RECV_1[34] := B#16#0;
   FC2_RECV_1[35] := B#16#0;
   FC2_RECV_1[36] := B#16#0;
   FC2_RECV_1[37] := B#16#0;
   FC2_RECV_1[38] := B#16#0;
   FC2_RECV_1[39] := B#16#0;
   FC2_RECV_1[40] := B#16#0;
   FC2_RECV_1[41] := B#16#0;
   FC2_RECV_1[42] := B#16#0;
   FC2_RECV_1[43] := B#16#0;
   FC2_RECV_1[44] := B#16#0;
   FC2_RECV_1[45] := B#16#0;
   FC2_RECV_1[46] := B#16#0;
   FC2_RECV_1[47] := B#16#0;
   FC2_RECV_1[48] := B#16#0;
   FC2_RECV_1[49] := B#16#0;
   FC2_RECV_1[50] := B#16#0;
   FC2_RECV_1[51] := B#16#0;
   FC2_RECV_1[52] := B#16#0;
   FC2_RECV_1[53] := B#16#0;
   FC2_RECV_1[54] := B#16#0;
   FC2_RECV_1[55] := B#16#0;
   FC2_RECV_1[56] := B#16#0;
   FC2_RECV_1[57] := B#16#0;
   FC2_RECV_1[58] := B#16#0;
   FC2_RECV_1[59] := B#16#0;
   FC2_RECV_1[60] := B#16#0;
   FC2_RECV_1[61] := B#16#0;
   FC2_RECV_1[62] := B#16#0;
   FC2_RECV_1[63] := B#16#0;
   FC2_RECV_1[64] := B#16#0;
   FC2_RECV_1[65] := B#16#0;
   FC2_RECV_1[66] := B#16#0;
   FC2_RECV_1[67] := B#16#0;
   FC2_RECV_1[68] := B#16#0;
   FC2_RECV_1[69] := B#16#0;
   FC2_RECV_1[70] := B#16#0;
   FC2_RECV_1[71] := B#16#0;
   FC2_RECV_1[72] := B#16#0;
   FC2_RECV_1[73] := B#16#0;
   FC2_RECV_1[74] := B#16#0;
   FC2_RECV_1[75] := B#16#0;
   FC2_RECV_1[76] := B#16#0;
   FC2_RECV_1[77] := B#16#0;
   FC2_RECV_1[78] := B#16#0;
   FC2_RECV_1[79] := B#16#0;
   FC2_RECV_1[80] := B#16#0;
   FC2_RECV_1[81] := B#16#0;
   FC2_RECV_1[82] := B#16#0;
   FC2_RECV_1[83] := B#16#0;
   FC2_RECV_1[84] := B#16#0;
   FC2_RECV_1[85] := B#16#0;
   FC2_RECV_1[86] := B#16#0;
   FC2_RECV_1[87] := B#16#0;
   FC2_RECV_1[88] := B#16#0;
   FC2_RECV_1[89] := B#16#0;
   FC2_RECV_1[90] := B#16#0;
   FC2_RECV_1[91] := B#16#0;
   FC2_RECV_1[92] := B#16#0;
   FC2_RECV_1[93] := B#16#0;
   FC2_RECV_1[94] := B#16#0;
   FC2_RECV_1[95] := B#16#0;
   FC2_RECV_1[96] := B#16#0;
   FC2_RECV_1[97] := B#16#0;
   FC2_RECV_1[98] := B#16#0;
   FC2_RECV_1[99] := B#16#0;
   FC2_RECV_1[100] := B#16#0;
   FC2_RECV_1[101] := B#16#0;
   FC2_RECV_1[102] := B#16#0;
   FC2_RECV_1[103] := B#16#0;
   FC2_RECV_1[104] := B#16#0;
   FC2_RECV_1[105] := B#16#0;
   FC2_RECV_1[106] := B#16#0;
   FC2_RECV_1[107] := B#16#0;
   FC2_RECV_1[108] := B#16#0;
   FC2_RECV_1[109] := B#16#0;
   FC2_RECV_1[110] := B#16#0;
   FC2_RECV_1[111] := B#16#0;
   FC2_RECV_1[112] := B#16#0;
   FC2_RECV_1[113] := B#16#0;
   FC2_RECV_1[114] := B#16#0;
   FC2_RECV_1[115] := B#16#0;
   FC2_RECV_1[116] := B#16#0;
   FC2_RECV_1[117] := B#16#0;
   FC2_RECV_1[118] := B#16#0;
   FC2_RECV_1[119] := B#16#0;
   FC2_RECV_1[120] := B#16#0;
   FC2_RECV_1[121] := B#16#0;
   FC2_RECV_1[122] := B#16#0;
   FC2_RECV_1[123] := B#16#0;
   FC2_RECV_1[124] := B#16#0;
   FC2_RECV_1[125] := B#16#0;
   FC2_RECV_1[126] := B#16#0;
   FC2_RECV_1[127] := B#16#0;
   FC2_RECV_1[128] := B#16#0;
   FC2_RECV_1[129] := B#16#0;
   FC2_RECV_1[130] := B#16#0;
   FC2_RECV_1[131] := B#16#0;
   FC2_RECV_1[132] := B#16#0;
   FC2_RECV_1[133] := B#16#0;
   FC2_RECV_1[134] := B#16#0;
   FC2_RECV_1[135] := B#16#0;
   FC2_RECV_1[136] := B#16#0;
   FC2_RECV_1[137] := B#16#0;
   FC2_RECV_1[138] := B#16#0;
   FC2_RECV_1[139] := B#16#0;
   FC2_RECV_1[140] := B#16#0;
   FC2_RECV_1[141] := B#16#0;
   FC2_RECV_1[142] := B#16#0;
   FC2_RECV_1[143] := B#16#0;
   FC2_RECV_1[144] := B#16#0;
   FC2_RECV_1[145] := B#16#0;
   FC2_RECV_1[146] := B#16#0;
   FC2_RECV_1[147] := B#16#0;
   FC2_RECV_1[148] := B#16#0;
   FC2_RECV_1[149] := B#16#0;
   FC2_RECV_1[150] := B#16#0;
   FC2_RECV_1[151] := B#16#0;
   FC2_RECV_1[152] := B#16#0;
   FC2_RECV_1[153] := B#16#0;
   FC2_RECV_1[154] := B#16#0;
   FC2_RECV_1[155] := B#16#0;
   FC2_RECV_1[156] := B#16#0;
   FC2_RECV_1[157] := B#16#0;
   FC2_RECV_1[158] := B#16#0;
   FC2_RECV_1[159] := B#16#0;
   FC2_RECV_1[160] := B#16#0;
   FC2_RECV_1[161] := B#16#0;
   FC2_RECV_1[162] := B#16#0;
   FC2_RECV_1[163] := B#16#0;
   FC2_RECV_1[164] := B#16#0;
   FC2_RECV_1[165] := B#16#0;
   FC2_RECV_1[166] := B#16#0;
   FC2_RECV_1[167] := B#16#0;
   FC2_RECV_1[168] := B#16#0;
   FC2_RECV_1[169] := B#16#0;
   FC2_RECV_1[170] := B#16#0;
   FC2_RECV_1[171] := B#16#0;
   FC2_RECV_1[172] := B#16#0;
   FC2_RECV_1[173] := B#16#0;
   FC2_RECV_1[174] := B#16#0;
   FC2_RECV_1[175] := B#16#0;
   FC2_RECV_1[176] := B#16#0;
   FC2_RECV_1[177] := B#16#0;
   FC2_RECV_1[178] := B#16#0;
   FC2_RECV_1[179] := B#16#0;
   FC2_RECV_1[180] := B#16#0;
   FC2_RECV_1[181] := B#16#0;
   FC2_RECV_1[182] := B#16#0;
   FC2_RECV_1[183] := B#16#0;
   FC2_RECV_1[184] := B#16#0;
   FC2_RECV_1[185] := B#16#0;
   FC2_RECV_1[186] := B#16#0;
   FC2_RECV_1[187] := B#16#0;
   FC2_RECV_1[188] := B#16#0;
   FC2_RECV_1[189] := B#16#0;
   FC2_RECV_1[190] := B#16#0;
   FC2_RECV_1[191] := B#16#0;
   FC2_RECV_1[192] := B#16#0;
   FC2_RECV_1[193] := B#16#0;
   FC2_RECV_1[194] := B#16#0;
   FC2_RECV_1[195] := B#16#0;
   FC2_RECV_1[196] := B#16#0;
   FC2_RECV_1[197] := B#16#0;
   FC2_RECV_1[198] := B#16#0;
   FC2_RECV_1[199] := B#16#0;
   FC2_RECV_1[200] := B#16#0;
   FC2_RECV_1[201] := B#16#0;
   FC2_RECV_1[202] := B#16#0;
   FC2_RECV_1[203] := B#16#0;
   FC2_RECV_1[204] := B#16#0;
   FC2_RECV_1[205] := B#16#0;
   FC2_RECV_1[206] := B#16#0;
   FC2_RECV_1[207] := B#16#0;
   FC2_RECV_1[208] := B#16#0;
   FC2_RECV_1[209] := B#16#0;
   FC2_RECV_1[210] := B#16#0;
   FC2_RECV_1[211] := B#16#0;
   FC2_RECV_1[212] := B#16#0;
   FC2_RECV_1[213] := B#16#0;
   FC2_RECV_1[214] := B#16#0;
   FC2_RECV_1[215] := B#16#0;
   FC2_RECV_1[216] := B#16#0;
   FC2_RECV_1[217] := B#16#0;
   FC2_RECV_1[218] := B#16#0;
   FC2_RECV_1[219] := B#16#0;
   FC2_RECV_1[220] := B#16#0;
   FC2_RECV_1[221] := B#16#0;
   FC2_RECV_1[222] := B#16#0;
   FC2_RECV_1[223] := B#16#0;
   FC2_RECV_1[224] := B#16#0;
   FC2_RECV_1[225] := B#16#0;
   FC2_RECV_1[226] := B#16#0;
   FC2_RECV_1[227] := B#16#0;
   FC2_RECV_1[228] := B#16#0;
   FC2_RECV_1[229] := B#16#0;
   FC2_RECV_1[230] := B#16#0;
   FC2_RECV_1[231] := B#16#0;
   FC2_RECV_1[232] := B#16#0;
   FC2_RECV_1[233] := B#16#0;
   FC2_RECV_1[234] := B#16#0;
   FC2_RECV_1[235] := B#16#0;
   FC2_RECV_1[236] := B#16#0;
   FC2_RECV_1[237] := B#16#0;
   FC2_RECV_1[238] := B#16#0;
   FC2_RECV_1[239] := B#16#0;
   FC2_RECV_1[240] := B#16#0;
   FC2_RECV_1[241] := B#16#0;
   FC2_RECV_1[242] := B#16#0;
   FC2_RECV_1[243] := B#16#0;
   FC2_RECV_1[244] := B#16#0;
   FC2_RECV_1[245] := B#16#0;
   FC2_RECV_1[246] := B#16#0;
   FC2_RECV_1[247] := B#16#0;
   FC2_RECV_1[248] := B#16#0;
   FC2_RECV_1[249] := B#16#0;
   FC2_RECV_1[250] := B#16#0;
   FC2_RECV_1[251] := B#16#0;
   FC2_RECV_1[252] := B#16#0;
   FC2_RECV_1[253] := B#16#0;
   FC2_RECV_1[254] := B#16#0;
   FC2_RECV_1[255] := B#16#0;
   FC2_RECV_1[256] := B#16#0;
   FC2_RECV_1[257] := B#16#0;
   FC2_RECV_1[258] := B#16#0;
   FC2_RECV_1[259] := B#16#0;
   FC2_RECV_1[260] := B#16#0;
   FC2_RECV_1[261] := B#16#0;
   FC2_RECV_1[262] := B#16#0;
   FC2_RECV_1[263] := B#16#0;
   FC2_RECV_1[264] := B#16#0;
   FC2_RECV_1[265] := B#16#0;
   FC2_RECV_1[266] := B#16#0;
   FC2_RECV_1[267] := B#16#0;
   FC2_RECV_1[268] := B#16#0;
   FC2_RECV_1[269] := B#16#0;
   FC2_RECV_1[270] := B#16#0;
   FC2_RECV_1[271] := B#16#0;
   FC2_RECV_1[272] := B#16#0;
   FC2_RECV_1[273] := B#16#0;
   FC2_RECV_1[274] := B#16#0;
   FC2_RECV_1[275] := B#16#0;
   FC2_RECV_1[276] := B#16#0;
   FC2_RECV_1[277] := B#16#0;
   FC2_RECV_1[278] := B#16#0;
   FC2_RECV_1[279] := B#16#0;
   FC2_RECV_1[280] := B#16#0;
   FC2_RECV_1[281] := B#16#0;
   FC2_RECV_1[282] := B#16#0;
   FC2_RECV_1[283] := B#16#0;
   FC2_RECV_1[284] := B#16#0;
   FC2_RECV_1[285] := B#16#0;
   FC2_RECV_1[286] := B#16#0;
   FC2_RECV_1[287] := B#16#0;
   FC2_RECV_1[288] := B#16#0;
   FC2_RECV_1[289] := B#16#0;
   FC2_RECV_1[290] := B#16#0;
   FC2_RECV_1[291] := B#16#0;
   FC2_RECV_1[292] := B#16#0;
   FC2_RECV_1[293] := B#16#0;
   FC2_RECV_1[294] := B#16#0;
   FC2_RECV_1[295] := B#16#0;
   FC2_RECV_1[296] := B#16#0;
   FC2_RECV_1[297] := B#16#0;
   FC2_RECV_1[298] := B#16#0;
   FC2_RECV_1[299] := B#16#0;
   FC2_RECV_1[300] := B#16#21;
   FC2_RECV_1[301] := B#16#0;
   FC2_RECV_1[302] := B#16#95;
   FC2_RECV_1[303] := B#16#AA;
   FC2_RECV_1[304] := B#16#EA;
   FC2_RECV_1[305] := B#16#FB;
   FC2_RECV_1[306] := B#16#EE;
   FC2_RECV_1[307] := B#16#F7;
   FC2_RECV_1[308] := B#16#AB;
   FC2_RECV_1[309] := B#16#22;
   FC2_RECV_1[310] := B#16#83;
   FC2_RECV_1[311] := B#16#AA;
   FC2_RECV_1[312] := B#16#0;
   FC2_RECV_1[313] := B#16#0;
   FC2_RECV_1[314] := B#16#0;
   FC2_RECV_1[315] := B#16#0;
   FC2_RECV_1[316] := B#16#0;
   FC2_RECV_1[317] := B#16#0;
   FC2_RECV_1[318] := B#16#0;
   FC2_RECV_1[319] := B#16#0;
   FC2_RECV_1[320] := B#16#0;
   FC2_RECV_1[321] := B#16#0;
   FC2_RECV_1[322] := B#16#0;
   FC2_RECV_1[323] := B#16#0;
   FC2_RECV_1[324] := B#16#0;
   FC2_RECV_1[325] := B#16#0;
   FC2_RECV_1[326] := B#16#0;
   FC2_RECV_1[327] := B#16#0;
   FC2_RECV_1[328] := B#16#0;
   FC2_RECV_1[329] := B#16#0;
   FC2_RECV_1[330] := B#16#0;
   FC2_RECV_1[331] := B#16#0;
   FC2_RECV_1[332] := B#16#0;
   FC2_RECV_1[333] := B#16#0;
   FC2_RECV_1[334] := B#16#0;
   FC2_RECV_1[335] := B#16#0;
   FC2_RECV_1[336] := B#16#0;
   FC2_RECV_1[337] := B#16#0;
   FC2_RECV_1[338] := B#16#0;
   FC2_RECV_1[339] := B#16#0;
   FC2_RECV_1[340] := B#16#0;
   FC2_RECV_1[341] := B#16#0;
   FC2_RECV_1[342] := B#16#0;
   FC2_RECV_1[343] := B#16#0;
   FC2_RECV_1[344] := B#16#0;
   FC2_RECV_1[345] := B#16#0;
   FC2_RECV_1[346] := B#16#0;
   FC2_RECV_1[347] := B#16#0;
   FC2_RECV_1[348] := B#16#0;
   FC2_RECV_1[349] := B#16#0;
   FC2_RECV_1[350] := B#16#0;
   FC2_RECV_1[351] := B#16#0;
   FC2_RECV_1[352] := B#16#0;
   FC2_RECV_1[353] := B#16#0;
   FC2_RECV_1[354] := B#16#0;
   FC2_RECV_1[355] := B#16#0;
   FC2_RECV_1[356] := B#16#0;
   FC2_RECV_1[357] := B#16#0;
   FC2_RECV_1[358] := B#16#0;
   FC2_RECV_1[359] := B#16#0;
   FC2_RECV_1[360] := B#16#0;
   FC2_RECV_1[361] := B#16#0;
   FC2_RECV_1[362] := B#16#0;
   FC2_RECV_1[363] := B#16#0;
   FC2_RECV_1[364] := B#16#0;
   FC2_RECV_1[365] := B#16#0;
   FC2_RECV_1[366] := B#16#0;
   FC2_RECV_1[367] := B#16#0;
   FC2_RECV_1[368] := B#16#0;
   FC2_RECV_1[369] := B#16#0;
   FC2_RECV_1[370] := B#16#0;
   FC2_RECV_1[371] := B#16#0;
   FC2_RECV_1[372] := B#16#0;
   FC2_RECV_1[373] := B#16#0;
   FC2_RECV_1[374] := B#16#0;
   FC2_RECV_1[375] := B#16#0;
   FC2_RECV_1[376] := B#16#0;
   FC2_RECV_1[377] := B#16#0;
   FC2_RECV_1[378] := B#16#0;
   FC2_RECV_1[379] := B#16#0;
   FC2_RECV_1[380] := B#16#0;
   FC2_RECV_1[381] := B#16#0;
   FC2_RECV_1[382] := B#16#0;
   FC2_RECV_1[383] := B#16#0;
   FC2_RECV_1[384] := B#16#0;
   FC2_RECV_1[385] := B#16#0;
   FC2_RECV_1[386] := B#16#0;
   FC2_RECV_1[387] := B#16#0;
   FC2_RECV_1[388] := B#16#0;
   FC2_RECV_1[389] := B#16#0;
   FC2_RECV_1[390] := B#16#0;
   FC2_RECV_1[391] := B#16#0;
   FC2_RECV_1[392] := B#16#0;
   FC2_RECV_1[393] := B#16#0;
   FC2_RECV_1[394] := B#16#0;
   FC2_RECV_1[395] := B#16#0;
   FC2_RECV_1[396] := B#16#0;
   FC2_RECV_1[397] := B#16#0;
   FC2_RECV_1[398] := B#16#0;
   FC2_RECV_1[399] := B#16#0;
   FC2_RECV_1[400] := B#16#0;
   FC2_RECV_1[401] := B#16#0;
   FC2_RECV_1[402] := B#16#0;
   FC2_RECV_1[403] := B#16#0;
   FC2_RECV_1[404] := B#16#0;
   FC2_RECV_1[405] := B#16#0;
   FC2_RECV_1[406] := B#16#0;
   FC2_RECV_1[407] := B#16#0;
   FC2_RECV_1[408] := B#16#0;
   FC2_RECV_1[409] := B#16#0;
   FC2_RECV_1[410] := B#16#0;
   FC2_RECV_1[411] := B#16#0;
   FC2_RECV_1[412] := B#16#0;
   FC2_RECV_1[413] := B#16#0;
   FC2_RECV_1[414] := B#16#0;
   FC2_RECV_1[415] := B#16#0;
   FC2_RECV_1[416] := B#16#0;
   FC2_RECV_1[417] := B#16#0;
   FC2_RECV_1[418] := B#16#0;
   FC2_RECV_1[419] := B#16#0;
   FC2_RECV_1[420] := B#16#0;
   FC2_RECV_1[421] := B#16#0;
   FC2_RECV_1[422] := B#16#0;
   FC2_RECV_1[423] := B#16#0;
   FC2_RECV_1[424] := B#16#0;
   FC2_RECV_1[425] := B#16#0;
   FC2_RECV_1[426] := B#16#0;
   FC2_RECV_1[427] := B#16#0;
   FC2_RECV_1[428] := B#16#0;
   FC2_RECV_1[429] := B#16#0;
   FC2_RECV_1[430] := B#16#0;
   FC2_RECV_1[431] := B#16#0;
   FC2_RECV_1[432] := B#16#0;
   FC2_RECV_1[433] := B#16#0;
   FC2_RECV_1[434] := B#16#0;
   FC2_RECV_1[435] := B#16#0;
   FC2_RECV_1[436] := B#16#0;
   FC2_RECV_1[437] := B#16#0;
   FC2_RECV_1[438] := B#16#0;
   FC2_RECV_1[439] := B#16#0;
   FC2_RECV_1[440] := B#16#0;
   FC2_RECV_1[441] := B#16#0;
   FC2_RECV_1[442] := B#16#0;
   FC2_RECV_1[443] := B#16#0;
   FC2_RECV_1[444] := B#16#0;
   FC2_RECV_1[445] := B#16#0;
   FC2_RECV_1[446] := B#16#0;
   FC2_RECV_1[447] := B#16#0;
   FC2_RECV_1[448] := B#16#0;
   FC2_RECV_1[449] := B#16#0;
   FC2_RECV_1[450] := B#16#0;
   FC2_RECV_1[451] := B#16#0;
   FC2_RECV_1[452] := B#16#0;
   FC2_RECV_1[453] := B#16#0;
   FC2_RECV_1[454] := B#16#0;
   FC2_RECV_1[455] := B#16#0;
   FC2_RECV_1[456] := B#16#0;
   FC2_RECV_1[457] := B#16#0;
   FC2_RECV_1[458] := B#16#0;
   FC2_RECV_1[459] := B#16#0;
   FC2_RECV_1[460] := B#16#0;
   FC2_RECV_1[461] := B#16#0;
   FC2_RECV_1[462] := B#16#0;
   FC2_RECV_1[463] := B#16#0;
   FC2_RECV_1[464] := B#16#0;
   FC2_RECV_1[465] := B#16#0;
   FC2_RECV_1[466] := B#16#0;
   FC2_RECV_1[467] := B#16#0;
   FC2_RECV_1[468] := B#16#0;
   FC2_RECV_1[469] := B#16#0;
   FC2_RECV_1[470] := B#16#0;
   FC2_RECV_1[471] := B#16#0;
   FC2_RECV_1[472] := B#16#0;
   FC2_RECV_1[473] := B#16#0;
   FC2_RECV_1[474] := B#16#0;
   FC2_RECV_1[475] := B#16#0;
   FC2_RECV_1[476] := B#16#0;
   FC2_RECV_1[477] := B#16#0;
   FC2_RECV_1[478] := B#16#0;
   FC2_RECV_1[479] := B#16#0;
   FC2_RECV_1[480] := B#16#0;
   FC2_RECV_1[481] := B#16#0;
   FC2_RECV_1[482] := B#16#0;
   FC2_RECV_1[483] := B#16#0;
   FC2_RECV_1[484] := B#16#0;
   FC2_RECV_1[485] := B#16#0;
   FC2_RECV_1[486] := B#16#0;
   FC2_RECV_1[487] := B#16#0;
   FC2_RECV_1[488] := B#16#0;
   FC2_RECV_1[489] := B#16#0;
   FC2_RECV_1[490] := B#16#0;
   FC2_RECV_1[491] := B#16#0;
   FC2_RECV_1[492] := B#16#0;
   FC2_RECV_1[493] := B#16#0;
   FC2_RECV_1[494] := B#16#0;
   FC2_RECV_1[495] := B#16#0;
   FC2_RECV_1[496] := B#16#0;
   FC2_RECV_1[497] := B#16#0;
   FC2_RECV_1[498] := B#16#0;
   FC2_RECV_1[499] := B#16#0;
END_DATA_BLOCK

DATA_BLOCK DB 62
TITLE =
VERSION : 0.1


